LIN {X 0,Y 324.336,Z 494.731,A -85,B 0,C 180,E1 -26772.496,E2 -26772.496} C_VEL
LIN {X 0,Y 334.682,Z 439.584,A -85,B 0,C 180,E1 -26774.316,E2 -26774.316} C_VEL
LIN {X 0,Y 333.314,Z 436.436,A -85,B 0,C 180,E1 -26776.094,E2 -26776.094} C_VEL
LIN {X 0,Y 331.956,Z 433.665,A -85,B 0,C 180,E1 -26778.901,E2 -26778.901} C_VEL
LIN {X 0,Y 331.571,Z 433.329,A -85,B 0,C 180,E1 -26780.673,E2 -26780.673} C_VEL
LIN {X 0,Y 331.565,Z 434.08,A -85,B 0,C 180,E1 -26782.586,E2 -26782.586} C_VEL
LIN {X 0,Y 332.161,Z 436.38,A -85,B 0,C 180,E1 -26784.82,E2 -26784.82} C_VEL
LIN {X 0,Y 333.09,Z 439.465,A -85,B 0,C 180,E1 -26786.646,E2 -26786.646} C_VEL
LIN {X 0,Y 334.002,Z 442.99,A -85,B 0,C 180,E1 -26788.056,E2 -26788.056} C_VEL
LIN {X 0,Y 324.195,Z 494.799,A -85,B 0,C 180,E1 -26789.774,E2 -26789.774} C_VEL
LIN {X 0,Y 320.598,Z 508.539,A -85,B 0,C 180,E1 -26790.375,E2 -26790.375} C_VEL
LIN {X 0,Y 316.075,Z 522.357,A -85,B 0,C 180,E1 -26791.184,E2 -26791.184} C_VEL
LIN {X 0,Y 310.686,Z 536.131,A -85,B 0,C 180,E1 -26792.248,E2 -26792.248} C_VEL
LIN {X 0,Y 304.524,Z 549.185,A -85,B 0,C 180,E1 -26793.534,E2 -26793.534} C_VEL
LIN {X 0,Y 298.181,Z 560.797,A -85,B 0,C 180,E1 -26794.987,E2 -26794.987} C_VEL
LIN {X 0,Y 291.665,Z 571.301,A -85,B 0,C 180,E1 -26796.649,E2 -26796.649} C_VEL
LIN {X 0,Y 285.414,Z 580.164,A -85,B 0,C 180,E1 -26798.4,E2 -26798.4} C_VEL
LIN {X 0,Y 278.653,Z 588.74,A -85,B 0,C 180,E1 -26800.545,E2 -26800.545} C_VEL
LIN {X 0,Y 272.465,Z 595.688,A -85,B 0,C 180,E1 -26802.804,E2 -26802.804} C_VEL
LIN {X 0,Y 266.016,Z 601.972,A -85,B 0,C 180,E1 -26805.514,E2 -26805.514} C_VEL
LIN {X 0,Y 260.17,Z 606.737,A -85,B 0,C 180,E1 -26808.351,E2 -26808.351} C_VEL
LIN {X 0,Y 255.014,Z 610.15,A -85,B 0,C 180,E1 -26811.439,E2 -26811.439} C_VEL
LIN {X 0,Y 252.065,Z 611.627,A -85,B 0,C 180,E1 -26813.618,E2 -26813.618} C_VEL
LIN {X 0,Y 248.579,Z 612.578,A -85,B 0,C 180,E1 -26816.769,E2 -26816.769} C_VEL
LIN {X 0,Y 246.132,Z 612.235,A -85,B 0,C 180,E1 -26820,E2 -26820} C_VEL
LIN {X 0,Y 244.401,Z 610.599,A -85,B 0,C 180,E1 -26823.286,E2 -26823.286} C_VEL
LIN {X 0,Y 243.306,Z 607.613,A -85,B 0,C 180,E1 -26826.612,E2 -26826.612} C_VEL
LIN {X 0,Y 243,Z 603.197,A -85,B 0,C 180,E1 -26829.959,E2 -26829.959} C_VEL
LIN {X 0,Y 242.985,Z 598.806,A -85,B 0,C 180,E1 -26832.486,E2 -26832.486} C_VEL
LIN {X 0,Y 243.239,Z 592.317,A -85,B 0,C 180,E1 -26835.448,E2 -26835.448} C_VEL
LIN {X 0,Y 243.619,Z 584.079,A -85,B 0,C 180,E1 -26838.437,E2 -26838.437} C_VEL
LIN {X 0,Y 244.159,Z 575.362,A -85,B 0,C 180,E1 -26841.014,E2 -26841.014} C_VEL
LIN {X 0,Y 244.883,Z 564.653,A -85,B 0,C 180,E1 -26843.606,E2 -26843.606} C_VEL
LIN {X 0,Y 245.783,Z 553.862,A -85,B 0,C 180,E1 -26845.76,E2 -26845.76} C_VEL
LIN {X 0,Y 246.865,Z 541.033,A -85,B 0,C 180,E1 -26847.87,E2 -26847.87} C_VEL
LIN {X 0,Y 247.927,Z 527.88,A -85,B 0,C 180,E1 -26849.631,E2 -26849.631} C_VEL
LIN {X 0,Y 249.014,Z 513.803,A -85,B 0,C 180,E1 -26851.122,E2 -26851.122} C_VEL
LIN {X 0,Y 250.108,Z 498.529,A -85,B 0,C 180,E1 -26852.359,E2 -26852.359} C_VEL
LIN {X 0,Y 251.001,Z 483.418,A -85,B 0,C 180,E1 -26853.241,E2 -26853.241} C_VEL
LIN {X 0,Y 255.021,Z 389.699,A -85,B 0,C 180,E1 -26857.363,E2 -26857.363} C_VEL
LIN {X 0,Y 252.513,Z 363.65,A -85,B 0,C 180,E1 -26858.616,E2 -26858.616} C_VEL
LIN {X 0,Y 251.535,Z 352.061,A -85,B 0,C 180,E1 -26859.176,E2 -26859.176} C_VEL
LIN {X 0,Y 250.283,Z 346.912,A -85,B 0,C 180,E1 -26859.516,E2 -26859.516} C_VEL
LIN {X 0,Y 246.827,Z 329.605,A -85,B 0,C 180,E1 -26863.64,E2 -26863.64} C_VEL
LIN {X 0,Y 246.163,Z 326.374,A -85,B 0,C 180,E1 -26864.432,E2 -26864.432} C_VEL
LIN {X 0,Y 246.097,Z 326.384,A -85,B 0,C 180,E1 -26869.104,E2 -26869.104} C_VEL
LIN {X 0,Y 246.107,Z 326.385,A -85,B 0,C 180,E1 -26873.292,E2 -26873.292} C_VEL
LIN {X 0,Y 246.115,Z 326.372,A -85,B 0,C 180,E1 -26877.262,E2 -26877.262} C_VEL
LIN {X 0,Y 246.14,Z 326.368,A -85,B 0,C 180,E1 -26881.906,E2 -26881.906} C_VEL
LIN {X 0,Y 246.192,Z 326.378,A -85,B 0,C 180,E1 -26886.523,E2 -26886.523} C_VEL
LIN {X 0,Y 246.258,Z 326.518,A -85,B 0,C 180,E1 -26887.721,E2 -26887.721} C_VEL
LIN {X 0,Y 247.292,Z 329.319,A -85,B 0,C 180,E1 -26887.949,E2 -26887.949} C_VEL
LIN {X 0,Y 255.224,Z 344.588,A -85,B 0,C 180,E1 -26889.436,E2 -26889.436} C_VEL
LIN {X 0,Y 263.934,Z 364.446,A -85,B 0,C 180,E1 -26891.038,E2 -26891.038} C_VEL
LIN {X 0,Y 264.785,Z 366.831,A -85,B 0,C 180,E1 -26891.201,E2 -26891.201} C_VEL
LIN {X 0,Y 261.589,Z 454.014,A -85,B 0,C 180,E1 -26893.517,E2 -26893.517} C_VEL
LIN {X 0,Y 260.624,Z 467.692,A -85,B 0,C 180,E1 -26894.156,E2 -26894.156} C_VEL
LIN {X 0,Y 259.477,Z 480.564,A -85,B 0,C 180,E1 -26895.037,E2 -26895.037} C_VEL
LIN {X 0,Y 257.894,Z 493.809,A -85,B 0,C 180,E1 -26896.248,E2 -26896.248} C_VEL
LIN {X 0,Y 256.075,Z 505.205,A -85,B 0,C 180,E1 -26897.557,E2 -26897.557} C_VEL
LIN {X 0,Y 253.893,Z 517.109,A -85,B 0,C 180,E1 -26899.264,E2 -26899.264} C_VEL
LIN {X 0,Y 251.992,Z 527.921,A -85,B 0,C 180,E1 -26901.202,E2 -26901.202} C_VEL
LIN {X 0,Y 250.122,Z 537.025,A -85,B 0,C 180,E1 -26903.161,E2 -26903.161} C_VEL
LIN {X 0,Y 248.243,Z 546.151,A -85,B 0,C 180,E1 -26905.546,E2 -26905.546} C_VEL
LIN {X 0,Y 246.553,Z 553.781,A -85,B 0,C 180,E1 -26907.961,E2 -26907.961} C_VEL
LIN {X 0,Y 245.444,Z 561.092,A -85,B 0,C 180,E1 -26910.849,E2 -26910.849} C_VEL
LIN {X 0,Y 244.645,Z 566.113,A -85,B 0,C 180,E1 -26913.279,E2 -26913.279} C_VEL
LIN {X 0,Y 243.723,Z 571.419,A -85,B 0,C 180,E1 -26916.597,E2 -26916.597} C_VEL
LIN {X 0,Y 243.365,Z 575.2,A -85,B 0,C 180,E1 -26919.94,E2 -26919.94} C_VEL
LIN {X 0,Y 243.416,Z 576.779,A -85,B 0,C 180,E1 -26921.938,E2 -26921.938} C_VEL
LIN {X 0,Y 243.611,Z 578.262,A -85,B 0,C 180,E1 -26924.993,E2 -26924.993} C_VEL
LIN {X 0,Y 244.447,Z 578.607,A -85,B 0,C 180,E1 -26928.368,E2 -26928.368} C_VEL
LIN {X 0,Y 245.791,Z 577.592,A -85,B 0,C 180,E1 -26931.74,E2 -26931.74} C_VEL
LIN {X 0,Y 247.865,Z 575.178,A -85,B 0,C 180,E1 -26935.075,E2 -26935.075} C_VEL
LIN {X 0,Y 250.574,Z 571.251,A -85,B 0,C 180,E1 -26938.368,E2 -26938.368} C_VEL
LIN {X 0,Y 253.98,Z 565.673,A -85,B 0,C 180,E1 -26941.596,E2 -26941.596} C_VEL
LIN {X 0,Y 257.568,Z 559.306,A -85,B 0,C 180,E1 -26944.348,E2 -26944.348} C_VEL
LIN {X 0,Y 261.631,Z 551.305,A -85,B 0,C 180,E1 -26947.035,E2 -26947.035} C_VEL
LIN {X 0,Y 265.504,Z 542.866,A -85,B 0,C 180,E1 -26949.278,E2 -26949.278} C_VEL
LIN {X 0,Y 269.799,Z 532.633,A -85,B 0,C 180,E1 -26951.448,E2 -26951.448} C_VEL
LIN {X 0,Y 273.597,Z 522.235,A -85,B 0,C 180,E1 -26953.217,E2 -26953.217} C_VEL
LIN {X 0,Y 277.182,Z 510.885,A -85,B 0,C 180,E1 -26954.776,E2 -26954.776} C_VEL
LIN {X 0,Y 280.433,Z 498.58,A -85,B 0,C 180,E1 -26956.123,E2 -26956.123} C_VEL
LIN {X 0,Y 283.166,Z 485.53,A -85,B 0,C 180,E1 -26957.247,E2 -26957.247} C_VEL
LIN {X 0,Y 285.407,Z 471.872,A -85,B 0,C 180,E1 -26958.12,E2 -26958.12} C_VEL
LIN {X 0,Y 286.998,Z 457.659,A -85,B 0,C 180,E1 -26958.759,E2 -26958.759} C_VEL
LIN {X 0,Y 288.327,Z 435.678,A -85,B 0,C 180,E1 -26959.349,E2 -26959.349} C_VEL
LIN {X 0,Y 290.593,Z 394.903,A -85,B 0,C 180,E1 -26960.299,E2 -26960.299} C_VEL
LIN {X 0,Y 285.026,Z 383.377,A -85,B 0,C 180,E1 -26961.787,E2 -26961.787} C_VEL
LIN {X 0,Y 277.938,Z 371.273,A -85,B 0,C 180,E1 -26963.732,E2 -26963.732} C_VEL
LIN {X 0,Y 269.772,Z 358.534,A -85,B 0,C 180,E1 -26966.163,E2 -26966.163} C_VEL
LIN {X 0,Y 263.662,Z 349.923,A -85,B 0,C 180,E1 -26968.131,E2 -26968.131} C_VEL
LIN {X 0,Y 260.517,Z 345.727,A -85,B 0,C 180,E1 -26969.206,E2 -26969.206} C_VEL
LIN {X 0,Y 257.438,Z 341.575,A -85,B 0,C 180,E1 -26970.314,E2 -26970.314} C_VEL
LIN {X 0,Y 254.794,Z 338.233,A -85,B 0,C 180,E1 -26971.303,E2 -26971.303} C_VEL
LIN {X 0,Y 253.958,Z 336.946,A -85,B 0,C 180,E1 -26971.637,E2 -26971.637} C_VEL
LIN {X 0,Y 251.405,Z 334.263,A -85,B 0,C 180,E1 -26972.626,E2 -26972.626} C_VEL
LIN {X 0,Y 250.075,Z 331.865,A -85,B 0,C 180,E1 -26973.211,E2 -26973.211} C_VEL
LIN {X 0,Y 247.587,Z 329.867,A -85,B 0,C 180,E1 -26974.216,E2 -26974.216} C_VEL
LIN {X 0,Y 246.353,Z 327.371,A -85,B 0,C 180,E1 -26974.818,E2 -26974.818} C_VEL
LIN {X 0,Y 246.153,Z 326.379,A -85,B 0,C 180,E1 -26974.985,E2 -26974.985} C_VEL
LIN {X 0,Y 246.241,Z 326.357,A -85,B 0,C 180,E1 -26980.041,E2 -26980.041} C_VEL
LIN {X 0,Y 246.352,Z 326.338,A -85,B 0,C 180,E1 -26985.173,E2 -26985.173} C_VEL
LIN {X 0,Y 246.419,Z 326.329,A -85,B 0,C 180,E1 -26990.18,E2 -26990.18} C_VEL
LIN {X 0,Y 246.664,Z 326.319,A -85,B 0,C 180,E1 -26993.616,E2 -26993.616} C_VEL
LIN {X 0,Y 246.74,Z 326.284,A -85,B 0,C 180,E1 -26996.745,E2 -26996.745} C_VEL
LIN {X 0,Y 246.882,Z 326.281,A -85,B 0,C 180,E1 -27000,E2 -27000} C_VEL
LIN {X 0,Y 246.676,Z 326.314,A -85,B 0,C 180,E1 -27004.887,E2 -27004.887} C_VEL
LIN {X 0,Y 246.504,Z 326.314,A -85,B 0,C 180,E1 -27008.168,E2 -27008.168} C_VEL
LIN {X 0,Y 246.377,Z 326.328,A -85,B 0,C 180,E1 -27013.146,E2 -27013.146} C_VEL
LIN {X 0,Y 246.238,Z 326.35,A -85,B 0,C 180,E1 -27016.527,E2 -27016.527} C_VEL
LIN {X 0,Y 246.239,Z 326.367,A -85,B 0,C 180,E1 -27020.178,E2 -27020.178} C_VEL
LIN {X 0,Y 246.182,Z 326.378,A -85,B 0,C 180,E1 -27024.441,E2 -27024.441} C_VEL
LIN {X 0,Y 246.116,Z 326.383,A -85,B 0,C 180,E1 -27028.935,E2 -27028.935} C_VEL
LIN {X 0,Y 246.158,Z 326.575,A -85,B 0,C 180,E1 -27030.337,E2 -27030.337} C_VEL
LIN {X 0,Y 248.112,Z 332.099,A -85,B 0,C 180,E1 -27034.376,E2 -27034.376} C_VEL
LIN {X 0,Y 249.773,Z 337.188,A -85,B 0,C 180,E1 -27037.671,E2 -27037.671} C_VEL
LIN {X 0,Y 250.499,Z 339.036,A -85,B 0,C 180,E1 -27038.421,E2 -27038.421} C_VEL
LIN {X 0,Y 252.088,Z 343.111,A -85,B 0,C 180,E1 -27039.303,E2 -27039.303} C_VEL
LIN {X 0,Y 255.959,Z 356.555,A -85,B 0,C 180,E1 -27041.169,E2 -27041.169} C_VEL
LIN {X 0,Y 257.972,Z 360.99,A -85,B 0,C 180,E1 -27041.993,E2 -27041.993} C_VEL
LIN {X 0,Y 262.83,Z 369.266,A -85,B 0,C 180,E1 -27043.728,E2 -27043.728} C_VEL
LIN {X 0,Y 269.015,Z 380.503,A -85,B 0,C 180,E1 -27045.79,E2 -27045.79} C_VEL
LIN {X 0,Y 275.663,Z 394.149,A -85,B 0,C 180,E1 -27047.871,E2 -27047.871} C_VEL
LIN {X 0,Y 281.475,Z 407.899,A -85,B 0,C 180,E1 -27049.612,E2 -27049.612} C_VEL
LIN {X 0,Y 283.693,Z 427.748,A -85,B 0,C 180,E1 -27050.754,E2 -27050.754} C_VEL
LIN {X 0,Y 280.723,Z 478.618,A -85,B 0,C 180,E1 -27051.981,E2 -27051.981} C_VEL
LIN {X 0,Y 278.945,Z 493.561,A -85,B 0,C 180,E1 -27052.55,E2 -27052.55} C_VEL
LIN {X 0,Y 276.399,Z 507.618,A -85,B 0,C 180,E1 -27053.342,E2 -27053.342} C_VEL
LIN {X 0,Y 273.137,Z 520.704,A -85,B 0,C 180,E1 -27054.314,E2 -27054.314} C_VEL
LIN {X 0,Y 269.411,Z 533.352,A -85,B 0,C 180,E1 -27055.569,E2 -27055.569} C_VEL
LIN {X 0,Y 265.436,Z 544.887,A -85,B 0,C 180,E1 -27057.031,E2 -27057.031} C_VEL
LIN {X 0,Y 261.709,Z 554.52,A -85,B 0,C 180,E1 -27058.545,E2 -27058.545} C_VEL
LIN {X 0,Y 257.195,Z 565.227,A -85,B 0,C 180,E1 -27060.65,E2 -27060.65} C_VEL
LIN {X 0,Y 252.953,Z 574.104,A -85,B 0,C 180,E1 -27062.818,E2 -27062.818} C_VEL
LIN {X 0,Y 248.616,Z 582.646,A -85,B 0,C 180,E1 -27065.45,E2 -27065.45} C_VEL
LIN {X 0,Y 244.877,Z 589.57,A -85,B 0,C 180,E1 -27068.175,E2 -27068.175} C_VEL
LIN {X 0,Y 241.579,Z 595.839,A -85,B 0,C 180,E1 -27071.406,E2 -27071.406} C_VEL
LIN {X 0,Y 239.033,Z 600.505,A -85,B 0,C 180,E1 -27074.713,E2 -27074.713} C_VEL
LIN {X 0,Y 237.261,Z 603.739,A -85,B 0,C 180,E1 -27078.078,E2 -27078.078} C_VEL
LIN {X 0,Y 236.26,Z 605.64,A -85,B 0,C 180,E1 -27081.48,E2 -27081.48} C_VEL
LIN {X 0,Y 236.139,Z 606.252,A -85,B 0,C 180,E1 -27084.899,E2 -27084.899} C_VEL
LIN {X 0,Y 236.758,Z 605.572,A -85,B 0,C 180,E1 -27088.309,E2 -27088.309} C_VEL
LIN {X 0,Y 236.863,Z 605.464,A -85,B 0,C 180,E1 -27088.839,E2 -27088.839} C_VEL
LIN {X 0,Y 236.642,Z 610.52,A -85,B 0,C 180,E1 -27091.7,E2 -27091.7} C_VEL
LIN {X 0,Y 236.296,Z 614.967,A -85,B 0,C 180,E1 -27095.106,E2 -27095.106} C_VEL
LIN {X 0,Y 236.54,Z 617.99,A -85,B 0,C 180,E1 -27098.519,E2 -27098.519} C_VEL
LIN {X 0,Y 237.781,Z 619.728,A -85,B 0,C 180,E1 -27101.904,E2 -27101.904} C_VEL
LIN {X 0,Y 240.003,Z 620.221,A -85,B 0,C 180,E1 -27105.232,E2 -27105.232} C_VEL
LIN {X 0,Y 243.059,Z 619.47,A -85,B 0,C 180,E1 -27108.485,E2 -27108.485} C_VEL
LIN {X 0,Y 247.046,Z 617.486,A -85,B 0,C 180,E1 -27111.632,E2 -27111.632} C_VEL
LIN {X 0,Y 252.05,Z 614.222,A -85,B 0,C 180,E1 -27114.64,E2 -27114.64} C_VEL
LIN {X 0,Y 257.622,Z 609.641,A -85,B 0,C 180,E1 -27117.534,E2 -27117.534} C_VEL
LIN {X 0,Y 264.117,Z 603.567,A -85,B 0,C 180,E1 -27120.261,E2 -27120.261} C_VEL
LIN {X 0,Y 271.466,Z 595.842,A -85,B 0,C 180,E1 -27122.813,E2 -27122.813} C_VEL
LIN {X 0,Y 278.383,Z 587.587,A -85,B 0,C 180,E1 -27124.923,E2 -27124.923} C_VEL
LIN {X 0,Y 285.87,Z 577.594,A -85,B 0,C 180,E1 -27126.895,E2 -27126.895} C_VEL
LIN {X 0,Y 292.736,Z 567.286,A -85,B 0,C 180,E1 -27128.474,E2 -27128.474} C_VEL
LIN {X 0,Y 299.238,Z 556.134,A -85,B 0,C 180,E1 -27129.854,E2 -27129.854} C_VEL
LIN {X 0,Y 305.485,Z 543.891,A -85,B 0,C 180,E1 -27131.025,E2 -27131.025} C_VEL
LIN {X 0,Y 311.332,Z 530.596,A -85,B 0,C 180,E1 -27132.018,E2 -27132.018} C_VEL
LIN {X 0,Y 316.265,Z 517.205,A -85,B 0,C 180,E1 -27132.776,E2 -27132.776} C_VEL
LIN {X 0,Y 320.797,Z 501.723,A -85,B 0,C 180,E1 -27133.461,E2 -27133.461} C_VEL
LIN {X 0,Y 324.988,Z 481.781,A -85,B 0,C 180,E1 -27134.153,E2 -27134.153} C_VEL
LIN {X 0,Y 332.174,Z 444.696,A -85,B 0,C 180,E1 -27135.374,E2 -27135.374} C_VEL
LIN {X 0,Y 331.261,Z 442.694,A -85,B 0,C 180,E1 -27136.763,E2 -27136.763} C_VEL
LIN {X 0,Y 330.257,Z 440.394,A -85,B 0,C 180,E1 -27139.321,E2 -27139.321} C_VEL
LIN {X 0,Y 329.944,Z 440.521,A -85,B 0,C 180,E1 -27141.769,E2 -27141.769} C_VEL
LIN {X 0,Y 330.263,Z 442.496,A -85,B 0,C 180,E1 -27144.061,E2 -27144.061} C_VEL
LIN {X 0,Y 330.815,Z 444.6,A -85,B 0,C 180,E1 -27145.522,E2 -27145.522} C_VEL
LIN {X 0,Y 331.491,Z 447.394,A -85,B 0,C 180,E1 -27146.868,E2 -27146.868} C_VEL
LIN {X 0,Y 331.544,Z 447.912,A -85,B 0,C 180,E1 -27147.019,E2 -27147.019} C_VEL
LIN {X 0,Y 322.252,Z 495.042,A -85,B 0,C 180,E1 -27148.556,E2 -27148.556} C_VEL
LIN {X 0,Y 318.393,Z 509.201,A -85,B 0,C 180,E1 -27149.169,E2 -27149.169} C_VEL
LIN {X 0,Y 313.488,Z 523.557,A -85,B 0,C 180,E1 -27150.004,E2 -27150.004} C_VEL
LIN {X 0,Y 307.748,Z 537.416,A -85,B 0,C 180,E1 -27151.075,E2 -27151.075} C_VEL
LIN {X 0,Y 300.838,Z 551.253,A -85,B 0,C 180,E1 -27152.456,E2 -27152.456} C_VEL
LIN {X 0,Y 294.321,Z 562.449,A -85,B 0,C 180,E1 -27153.879,E2 -27153.879} C_VEL
LIN {X 0,Y 287.545,Z 572.735,A -85,B 0,C 180,E1 -27155.537,E2 -27155.537} C_VEL
LIN {X 0,Y 280.861,Z 581.621,A -85,B 0,C 180,E1 -27157.338,E2 -27157.338} C_VEL
LIN {X 0,Y 274.007,Z 589.691,A -85,B 0,C 180,E1 -27159.421,E2 -27159.421} C_VEL
LIN {X 0,Y 267.52,Z 596.488,A -85,B 0,C 180,E1 -27161.688,E2 -27161.688} C_VEL
LIN {X 0,Y 260.74,Z 602.634,A -85,B 0,C 180,E1 -27164.417,E2 -27164.417} C_VEL
LIN {X 0,Y 254.608,Z 607.263,A -85,B 0,C 180,E1 -27167.286,E2 -27167.286} C_VEL
LIN {X 0,Y 249.313,Z 610.449,A -85,B 0,C 180,E1 -27170.295,E2 -27170.295} C_VEL
LIN {X 0,Y 244.945,Z 612.283,A -85,B 0,C 180,E1 -27173.432,E2 -27173.432} C_VEL
LIN {X 0,Y 241.432,Z 612.82,A -85,B 0,C 180,E1 -27176.674,E2 -27176.674} C_VEL
LIN {X 0,Y 238.962,Z 612.075,A -85,B 0,C 180,E1 -27180,E2 -27180} C_VEL
LIN {X 0,Y 237.236,Z 610.044,A -85,B 0,C 180,E1 -27183.385,E2 -27183.385} C_VEL
LIN {X 0,Y 236.193,Z 606.65,A -85,B 0,C 180,E1 -27186.813,E2 -27186.813} C_VEL
LIN {X 0,Y 235.943,Z 601.793,A -85,B 0,C 180,E1 -27190.26,E2 -27190.26} C_VEL
LIN {X 0,Y 235.966,Z 597.046,A -85,B 0,C 180,E1 -27192.864,E2 -27192.864} C_VEL
LIN {X 0,Y 236.283,Z 590.09,A -85,B 0,C 180,E1 -27195.915,E2 -27195.915} C_VEL
LIN {X 0,Y 236.657,Z 582.174,A -85,B 0,C 180,E1 -27198.707,E2 -27198.707} C_VEL
LIN {X 0,Y 237.175,Z 573.576,A -85,B 0,C 180,E1 -27201.209,E2 -27201.209} C_VEL
LIN {X 0,Y 237.977,Z 562.146,A -85,B 0,C 180,E1 -27203.949,E2 -27203.949} C_VEL
LIN {X 0,Y 238.967,Z 550.077,A -85,B 0,C 180,E1 -27206.317,E2 -27206.317} C_VEL
LIN {X 0,Y 240.059,Z 537.136,A -85,B 0,C 180,E1 -27208.366,E2 -27208.366} C_VEL
LIN {X 0,Y 241.147,Z 523.888,A -85,B 0,C 180,E1 -27210.069,E2 -27210.069} C_VEL
LIN {X 0,Y 242.168,Z 509.966,A -85,B 0,C 180,E1 -27211.496,E2 -27211.496} C_VEL
LIN {X 0,Y 243.2,Z 495.468,A -85,B 0,C 180,E1 -27212.624,E2 -27212.624} C_VEL
LIN {X 0,Y 244.086,Z 479.061,A -85,B 0,C 180,E1 -27213.53,E2 -27213.53} C_VEL
LIN {X 0,Y 247.981,Z 390.378,A -85,B 0,C 180,E1 -27217.561,E2 -27217.561} C_VEL
LIN {X 0,Y 245.383,Z 362.456,A -85,B 0,C 180,E1 -27218.948,E2 -27218.948} C_VEL
LIN {X 0,Y 244.574,Z 353.328,A -85,B 0,C 180,E1 -27219.407,E2 -27219.407} C_VEL
LIN {X 0,Y 243.104,Z 347.07,A -85,B 0,C 180,E1 -27219.816,E2 -27219.816} C_VEL
LIN {X 0,Y 239.64,Z 329.856,A -85,B 0,C 180,E1 -27224.001,E2 -27224.001} C_VEL
LIN {X 0,Y 239.115,Z 327.25,A -85,B 0,C 180,E1 -27224.671,E2 -27224.671} C_VEL
LIN {X 0,Y 239.062,Z 327.259,A -85,B 0,C 180,E1 -27229.86,E2 -27229.86} C_VEL
LIN {X 0,Y 239.033,Z 327.258,A -85,B 0,C 180,E1 -27234.117,E2 -27234.117} C_VEL
LIN {X 0,Y 239.084,Z 327.256,A -85,B 0,C 180,E1 -27238.17,E2 -27238.17} C_VEL
LIN {X 0,Y 239.101,Z 327.244,A -85,B 0,C 180,E1 -27242.045,E2 -27242.045} C_VEL
LIN {X 0,Y 239.161,Z 327.274,A -85,B 0,C 180,E1 -27246.775,E2 -27246.775} C_VEL
LIN {X 0,Y 240.225,Z 330.204,A -85,B 0,C 180,E1 -27247.025,E2 -27247.025} C_VEL
LIN {X 0,Y 247.828,Z 344.438,A -85,B 0,C 180,E1 -27248.515,E2 -27248.515} C_VEL
LIN {X 0,Y 256.291,Z 363.144,A -85,B 0,C 180,E1 -27250.143,E2 -27250.143} C_VEL
LIN {X 0,Y 258.304,Z 368.174,A -85,B 0,C 180,E1 -27250.529,E2 -27250.529} C_VEL
LIN {X 0,Y 255.131,Z 454.419,A -85,B 0,C 180,E1 -27252.882,E2 -27252.882} C_VEL
LIN {X 0,Y 254.127,Z 468.101,A -85,B 0,C 180,E1 -27253.534,E2 -27253.534} C_VEL
LIN {X 0,Y 252.798,Z 482.095,A -85,B 0,C 180,E1 -27254.529,E2 -27254.529} C_VEL
LIN {X 0,Y 251.077,Z 495.959,A -85,B 0,C 180,E1 -27255.867,E2 -27255.867} C_VEL
LIN {X 0,Y 248.941,Z 508.449,A -85,B 0,C 180,E1 -27257.401,E2 -27257.401} C_VEL
LIN {X 0,Y 246.757,Z 519.848,A -85,B 0,C 180,E1 -27259.157,E2 -27259.157} C_VEL
LIN {X 0,Y 245.004,Z 529.301,A -85,B 0,C 180,E1 -27260.949,E2 -27260.949} C_VEL
LIN {X 0,Y 242.7,Z 539.876,A -85,B 0,C 180,E1 -27263.367,E2 -27263.367} C_VEL
LIN {X 0,Y 240.884,Z 548.588,A -85,B 0,C 180,E1 -27265.827,E2 -27265.827} C_VEL
LIN {X 0,Y 239.242,Z 555.863,A -85,B 0,C 180,E1 -27268.318,E2 -27268.318} C_VEL
LIN {X 0,Y 238.204,Z 562.68,A -85,B 0,C 180,E1 -27271.211,E2 -27271.211} C_VEL
LIN {X 0,Y 237.237,Z 568.335,A -85,B 0,C 180,E1 -27274.229,E2 -27274.229} C_VEL
LIN {X 0,Y 236.448,Z 573.187,A -85,B 0,C 180,E1 -27277.656,E2 -27277.656} C_VEL
LIN {X 0,Y 236.267,Z 575.802,A -85,B 0,C 180,E1 -27280.242,E2 -27280.242} C_VEL
LIN {X 0,Y 236.385,Z 578.103,A -85,B 0,C 180,E1 -27283.708,E2 -27283.708} C_VEL
LIN {X 0,Y 236.982,Z 579.048,A -85,B 0,C 180,E1 -27287.187,E2 -27287.187} C_VEL
LIN {X 0,Y 238.207,Z 578.633,A -85,B 0,C 180,E1 -27290.657,E2 -27290.657} C_VEL
LIN {X 0,Y 240.027,Z 576.841,A -85,B 0,C 180,E1 -27294.109,E2 -27294.109} C_VEL
LIN {X 0,Y 242.596,Z 573.572,A -85,B 0,C 180,E1 -27297.509,E2 -27297.509} C_VEL
LIN {X 0,Y 245.841,Z 568.734,A -85,B 0,C 180,E1 -27300.849,E2 -27300.849} C_VEL
LIN {X 0,Y 248.786,Z 564.008,A -85,B 0,C 180,E1 -27303.294,E2 -27303.294} C_VEL
LIN {X 0,Y 252.989,Z 556.513,A -85,B 0,C 180,E1 -27306.278,E2 -27306.278} C_VEL
LIN {X 0,Y 257.101,Z 548.39,A -85,B 0,C 180,E1 -27308.795,E2 -27308.795} C_VEL
LIN {X 0,Y 261.2,Z 539.516,A -85,B 0,C 180,E1 -27310.984,E2 -27310.984} C_VEL
LIN {X 0,Y 265.133,Z 530.093,A -85,B 0,C 180,E1 -27312.859,E2 -27312.859} C_VEL
LIN {X 0,Y 269.128,Z 519.084,A -85,B 0,C 180,E1 -27314.639,E2 -27314.639} C_VEL
LIN {X 0,Y 272.872,Z 506.946,A -85,B 0,C 180,E1 -27316.209,E2 -27316.209} C_VEL
LIN {X 0,Y 275.866,Z 495.22,A -85,B 0,C 180,E1 -27317.414,E2 -27317.414} C_VEL
LIN {X 0,Y 278.671,Z 481.327,A -85,B 0,C 180,E1 -27318.527,E2 -27318.527} C_VEL
LIN {X 0,Y 280.812,Z 467.022,A -85,B 0,C 180,E1 -27319.347,E2 -27319.347} C_VEL
LIN {X 0,Y 282.152,Z 453.648,A -85,B 0,C 180,E1 -27319.864,E2 -27319.864} C_VEL
LIN {X 0,Y 285.374,Z 397.385,A -85,B 0,C 180,E1 -27321.224,E2 -27321.224} C_VEL
LIN {X 0,Y 280.292,Z 386.884,A -85,B 0,C 180,E1 -27322.643,E2 -27322.643} C_VEL
LIN {X 0,Y 272.88,Z 374.249,A -85,B 0,C 180,E1 -27324.778,E2 -27324.778} C_VEL
LIN {X 0,Y 265.612,Z 362.906,A -85,B 0,C 180,E1 -27327.05,E2 -27327.05} C_VEL
LIN {X 0,Y 260.015,Z 355.002,A -85,B 0,C 180,E1 -27328.933,E2 -27328.933} C_VEL
LIN {X 0,Y 256.903,Z 350.768,A -85,B 0,C 180,E1 -27330.047,E2 -27330.047} C_VEL
LIN {X 0,Y 254.324,Z 347.231,A -85,B 0,C 180,E1 -27331.019,E2 -27331.019} C_VEL
LIN {X 0,Y 251.511,Z 343.38,A -85,B 0,C 180,E1 -27332.129,E2 -27332.129} C_VEL
LIN {X 0,Y 248.474,Z 339.882,A -85,B 0,C 180,E1 -27333.359,E2 -27333.359} C_VEL
LIN {X 0,Y 247.369,Z 338.074,A -85,B 0,C 180,E1 -27333.854,E2 -27333.854} C_VEL
LIN {X 0,Y 244.809,Z 335.604,A -85,B 0,C 180,E1 -27334.952,E2 -27334.952} C_VEL
LIN {X 0,Y 243.284,Z 332.858,A -85,B 0,C 180,E1 -27335.709,E2 -27335.709} C_VEL
LIN {X 0,Y 240.736,Z 330.955,A -85,B 0,C 180,E1 -27336.872,E2 -27336.872} C_VEL
LIN {X 0,Y 239.49,Z 328.827,A -85,B 0,C 180,E1 -27337.54,E2 -27337.54} C_VEL
LIN {X 0,Y 239.114,Z 327.246,A -85,B 0,C 180,E1 -27337.843,E2 -27337.843} C_VEL
LIN {X 0,Y 239.156,Z 327.233,A -85,B 0,C 180,E1 -27341.206,E2 -27341.206} C_VEL
LIN {X 0,Y 239.284,Z 327.219,A -85,B 0,C 180,E1 -27344.995,E2 -27344.995} C_VEL
LIN {X 0,Y 239.367,Z 327.209,A -85,B 0,C 180,E1 -27349.888,E2 -27349.888} C_VEL
LIN {X 0,Y 239.641,Z 327.193,A -85,B 0,C 180,E1 -27353.563,E2 -27353.563} C_VEL
LIN {X 0,Y 239.709,Z 327.159,A -85,B 0,C 180,E1 -27356.65,E2 -27356.65} C_VEL
LIN {X 0,Y 239.847,Z 327.157,A -85,B 0,C 180,E1 -27360,E2 -27360} C_VEL
LIN {X 0,Y 239.711,Z 327.167,A -85,B 0,C 180,E1 -27363.35,E2 -27363.35} C_VEL
LIN {X 0,Y 239.603,Z 327.172,A -85,B 0,C 180,E1 -27366.715,E2 -27366.715} C_VEL
LIN {X 0,Y 239.349,Z 327.204,A -85,B 0,C 180,E1 -27371.821,E2 -27371.821} C_VEL
LIN {X 0,Y 239.28,Z 327.233,A -85,B 0,C 180,E1 -27375.275,E2 -27375.275} C_VEL
LIN {X 0,Y 239.175,Z 327.241,A -85,B 0,C 180,E1 -27380.575,E2 -27380.575} C_VEL
LIN {X 0,Y 239.12,Z 327.254,A -85,B 0,C 180,E1 -27384.772,E2 -27384.772} C_VEL
LIN {X 0,Y 239.131,Z 327.352,A -85,B 0,C 180,E1 -27387.71,E2 -27387.71} C_VEL
LIN {X 0,Y 241.226,Z 333.465,A -85,B 0,C 180,E1 -27392.65,E2 -27392.65} C_VEL
LIN {X 0,Y 242.742,Z 337.837,A -85,B 0,C 180,E1 -27395.611,E2 -27395.611} C_VEL
LIN {X 0,Y 246.06,Z 342.861,A -85,B 0,C 180,E1 -27397.173,E2 -27397.173} C_VEL
LIN {X 0,Y 247.675,Z 344.955,A -85,B 0,C 180,E1 -27397.873,E2 -27397.873} C_VEL
LIN {X 0,Y 251.111,Z 350.075,A -85,B 0,C 180,E1 -27399.325,E2 -27399.325} C_VEL
LIN {X 0,Y 256.089,Z 357.941,A -85,B 0,C 180,E1 -27401.289,E2 -27401.289} C_VEL
LIN {X 0,Y 257.972,Z 360.99,A -85,B 0,C 180,E1 -27401.993,E2 -27401.993} C_VEL
LIN {X 0,Y 260.017,Z 365.229,A -85,B 0,C 180,E1 -27402.774,E2 -27402.774} C_VEL
LIN {X 0,Y 261.538,Z 370.158,A -85,B 0,C 180,E1 -27403.415,E2 -27403.415} C_VEL
LIN {X 0,Y 265.001,Z 384.136,A -85,B 0,C 180,E1 -27404.93,E2 -27404.93} C_VEL
LIN {X 0,Y 266.209,Z 387.353,A -85,B 0,C 180,E1 -27405.37,E2 -27405.37} C_VEL
LIN {X 0,Y 272.772,Z 401.414,A -85,B 0,C 180,E1 -27407.499,E2 -27407.499} C_VEL
LIN {X 0,Y 276.741,Z 411.518,A -85,B 0,C 180,E1 -27408.754,E2 -27408.754} C_VEL
LIN {X 0,Y 278.598,Z 429.253,A -85,B 0,C 180,E1 -27409.789,E2 -27409.789} C_VEL
LIN {X 0,Y 275.483,Z 479.381,A -85,B 0,C 180,E1 -27411.007,E2 -27411.007} C_VEL
LIN {X 0,Y 273.639,Z 493.819,A -85,B 0,C 180,E1 -27411.577,E2 -27411.577} C_VEL
LIN {X 0,Y 271.024,Z 507.702,A -85,B 0,C 180,E1 -27412.374,E2 -27412.374} C_VEL
LIN {X 0,Y 267.417,Z 521.559,A -85,B 0,C 180,E1 -27413.429,E2 -27413.429} C_VEL
LIN {X 0,Y 263.625,Z 533.958,A -85,B 0,C 180,E1 -27414.703,E2 -27414.703} C_VEL
LIN {X 0,Y 259.082,Z 546.483,A -85,B 0,C 180,E1 -27416.347,E2 -27416.347} C_VEL
LIN {X 0,Y 254.92,Z 556.747,A -85,B 0,C 180,E1 -27418.072,E2 -27418.072} C_VEL
LIN {X 0,Y 250.291,Z 567.002,A -85,B 0,C 180,E1 -27420.22,E2 -27420.22} C_VEL
LIN {X 0,Y 245.971,Z 575.519,A -85,B 0,C 180,E1 -27422.44,E2 -27422.44} C_VEL
LIN {X 0,Y 241.572,Z 583.701,A -85,B 0,C 180,E1 -27425.143,E2 -27425.143} C_VEL
LIN {X 0,Y 238.275,Z 589.47,A -85,B 0,C 180,E1 -27427.538,E2 -27427.538} C_VEL
LIN {X 0,Y 234.836,Z 595.651,A -85,B 0,C 180,E1 -27430.851,E2 -27430.851} C_VEL
LIN {X 0,Y 232.15,Z 600.243,A -85,B 0,C 180,E1 -27434.248,E2 -27434.248} C_VEL
LIN {X 0,Y 230.282,Z 603.42,A -85,B 0,C 180,E1 -27437.711,E2 -27437.711} C_VEL
LIN {X 0,Y 229.214,Z 605.265,A -85,B 0,C 180,E1 -27441.216,E2 -27441.216} C_VEL
LIN {X 0,Y 229.041,Z 605.821,A -85,B 0,C 180,E1 -27444.74,E2 -27444.74} C_VEL
LIN {X 0,Y 229.655,Z 605.086,A -85,B 0,C 180,E1 -27448.257,E2 -27448.257} C_VEL
LIN {X 0,Y 229.871,Z 604.838,A -85,B 0,C 180,E1 -27449.24,E2 -27449.24} C_VEL
LIN {X 0,Y 229.653,Z 609.278,A -85,B 0,C 180,E1 -27451.752,E2 -27451.752} C_VEL
LIN {X 0,Y 229.314,Z 613.971,A -85,B 0,C 180,E1 -27455.262,E2 -27455.262} C_VEL
LIN {X 0,Y 229.544,Z 617.232,A -85,B 0,C 180,E1 -27458.78,E2 -27458.78} C_VEL
LIN {X 0,Y 230.839,Z 619.23,A -85,B 0,C 180,E1 -27462.267,E2 -27462.267} C_VEL
LIN {X 0,Y 233.153,Z 619.992,A -85,B 0,C 180,E1 -27465.691,E2 -27465.691} C_VEL
LIN {X 0,Y 236.334,Z 619.526,A -85,B 0,C 180,E1 -27469.031,E2 -27469.031} C_VEL
LIN {X 0,Y 240.476,Z 617.84,A -85,B 0,C 180,E1 -27472.255,E2 -27472.255} C_VEL
LIN {X 0,Y 245.643,Z 614.89,A -85,B 0,C 180,E1 -27475.327,E2 -27475.327} C_VEL
LIN {X 0,Y 251.422,Z 610.655,A -85,B 0,C 180,E1 -27478.273,E2 -27478.273} C_VEL
LIN {X 0,Y 258.128,Z 605.007,A -85,B 0,C 180,E1 -27481.04,E2 -27481.04} C_VEL
LIN {X 0,Y 265.683,Z 597.785,A -85,B 0,C 180,E1 -27483.621,E2 -27483.621} C_VEL
LIN {X 0,Y 273.863,Z 588.755,A -85,B 0,C 180,E1 -27486.037,E2 -27486.037} C_VEL
LIN {X 0,Y 281.603,Z 579.054,A -85,B 0,C 180,E1 -27488.001,E2 -27488.001} C_VEL
LIN {X 0,Y 288.679,Z 569.115,A -85,B 0,C 180,E1 -27489.567,E2 -27489.567} C_VEL
LIN {X 0,Y 296.006,Z 557.336,A -85,B 0,C 180,E1 -27491.049,E2 -27491.049} C_VEL
LIN {X 0,Y 303.024,Z 544.289,A -85,B 0,C 180,E1 -27492.295,E2 -27492.295} C_VEL
LIN {X 0,Y 309.136,Z 530.975,A -85,B 0,C 180,E1 -27493.271,E2 -27493.271} C_VEL
LIN {X 0,Y 314.7,Z 516.399,A -85,B 0,C 180,E1 -27494.074,E2 -27494.074} C_VEL
LIN {X 0,Y 319.497,Z 500.196,A -85,B 0,C 180,E1 -27494.769,E2 -27494.769} C_VEL
LIN {X 0,Y 324.264,Z 477.875,A -85,B 0,C 180,E1 -27495.505,E2 -27495.505} C_VEL
LIN {X 0,Y 329.836,Z 450.121,A -85,B 0,C 180,E1 -27496.418,E2 -27496.418} C_VEL
LIN {X 0,Y 328.712,Z 447.44,A -85,B 0,C 180,E1 -27499.089,E2 -27499.089} C_VEL
LIN {X 0,Y 328.339,Z 447.28,A -85,B 0,C 180,E1 -27501.355,E2 -27501.355} C_VEL
LIN {X 0,Y 328.513,Z 448.861,A -85,B 0,C 180,E1 -27503.512,E2 -27503.512} C_VEL
LIN {X 0,Y 329.029,Z 451.267,A -85,B 0,C 180,E1 -27505.247,E2 -27505.247} C_VEL
LIN {X 0,Y 329.341,Z 452.534,A -85,B 0,C 180,E1 -27505.933,E2 -27505.933} C_VEL
LIN {X 0,Y 320.454,Z 495.837,A -85,B 0,C 180,E1 -27507.342,E2 -27507.342} C_VEL
LIN {X 0,Y 316.574,Z 509.532,A -85,B 0,C 180,E1 -27507.926,E2 -27507.926} C_VEL
LIN {X 0,Y 311.671,Z 523.409,A -85,B 0,C 180,E1 -27508.707,E2 -27508.707} C_VEL
LIN {X 0,Y 305.781,Z 537.184,A -85,B 0,C 180,E1 -27509.738,E2 -27509.738} C_VEL
LIN {X 0,Y 298.682,Z 550.935,A -85,B 0,C 180,E1 -27511.074,E2 -27511.074} C_VEL
LIN {X 0,Y 291.69,Z 562.494,A -85,B 0,C 180,E1 -27512.503,E2 -27512.503} C_VEL
LIN {X 0,Y 284.761,Z 572.61,A -85,B 0,C 180,E1 -27514.112,E2 -27514.112} C_VEL
LIN {X 0,Y 277.928,Z 581.311,A -85,B 0,C 180,E1 -27515.824,E2 -27515.824} C_VEL
LIN {X 0,Y 270.517,Z 589.662,A -85,B 0,C 180,E1 -27517.948,E2 -27517.948} C_VEL
LIN {X 0,Y 264.602,Z 595.615,A -85,B 0,C 180,E1 -27519.871,E2 -27519.871} C_VEL
LIN {X 0,Y 257.281,Z 602,A -85,B 0,C 180,E1 -27522.574,E2 -27522.574} C_VEL
LIN {X 0,Y 250.709,Z 606.813,A -85,B 0,C 180,E1 -27525.437,E2 -27525.437} C_VEL
LIN {X 0,Y 244.855,Z 610.209,A -85,B 0,C 180,E1 -27528.449,E2 -27528.449} C_VEL
LIN {X 0,Y 239.937,Z 612.251,A -85,B 0,C 180,E1 -27531.607,E2 -27531.607} C_VEL
LIN {X 0,Y 235.925,Z 612.999,A -85,B 0,C 180,E1 -27534.89,E2 -27534.89} C_VEL
LIN {X 0,Y 232.908,Z 612.472,A -85,B 0,C 180,E1 -27538.277,E2 -27538.277} C_VEL
LIN {X 0,Y 230.855,Z 610.682,A -85,B 0,C 180,E1 -27541.739,E2 -27541.739} C_VEL
LIN {X 0,Y 229.518,Z 607.574,A -85,B 0,C 180,E1 -27545.253,E2 -27545.253} C_VEL
LIN {X 0,Y 228.95,Z 603.063,A -85,B 0,C 180,E1 -27548.799,E2 -27548.799} C_VEL
LIN {X 0,Y 228.914,Z 598.174,A -85,B 0,C 180,E1 -27551.702,E2 -27551.702} C_VEL
LIN {X 0,Y 229.139,Z 591.032,A -85,B 0,C 180,E1 -27555.06,E2 -27555.06} C_VEL
LIN {X 0,Y 229.481,Z 583.816,A -85,B 0,C 180,E1 -27557.772,E2 -27557.772} C_VEL
LIN {X 0,Y 229.99,Z 575.054,A -85,B 0,C 180,E1 -27560.502,E2 -27560.502} C_VEL
LIN {X 0,Y 230.554,Z 566.247,A -85,B 0,C 180,E1 -27562.79,E2 -27562.79} C_VEL
LIN {X 0,Y 231.474,Z 554.62,A -85,B 0,C 180,E1 -27565.304,E2 -27565.304} C_VEL
LIN {X 0,Y 232.587,Z 541.7,A -85,B 0,C 180,E1 -27567.582,E2 -27567.582} C_VEL
LIN {X 0,Y 233.674,Z 528.697,A -85,B 0,C 180,E1 -27569.45,E2 -27569.45} C_VEL
LIN {X 0,Y 234.733,Z 515.442,A -85,B 0,C 180,E1 -27570.98,E2 -27570.98} C_VEL
LIN {X 0,Y 235.802,Z 500.327,A -85,B 0,C 180,E1 -27572.323,E2 -27572.323} C_VEL
LIN {X 0,Y 236.756,Z 485.061,A -85,B 0,C 180,E1 -27573.31,E2 -27573.31} C_VEL
LIN {X 0,Y 240.958,Z 391.001,A -85,B 0,C 180,E1 -27577.763,E2 -27577.763} C_VEL
LIN {X 0,Y 238.4,Z 363.366,A -85,B 0,C 180,E1 -27579.179,E2 -27579.179} C_VEL
LIN {X 0,Y 237.651,Z 354.55,A -85,B 0,C 180,E1 -27579.635,E2 -27579.635} C_VEL
LIN {X 0,Y 235.917,Z 347.305,A -85,B 0,C 180,E1 -27580.089,E2 -27580.089} C_VEL
LIN {X 0,Y 232.509,Z 330.339,A -85,B 0,C 180,E1 -27584.313,E2 -27584.313} C_VEL
LIN {X 0,Y 232.077,Z 328.125,A -85,B 0,C 180,E1 -27584.896,E2 -27584.896} C_VEL
LIN {X 0,Y 231.995,Z 328.141,A -85,B 0,C 180,E1 -27589.008,E2 -27589.008} C_VEL
LIN {X 0,Y 231.999,Z 328.143,A -85,B 0,C 180,E1 -27592.851,E2 -27592.851} C_VEL
LIN {X 0,Y 231.987,Z 328.128,A -85,B 0,C 180,E1 -27597.075,E2 -27597.075} C_VEL
LIN {X 0,Y 232.036,Z 328.127,A -85,B 0,C 180,E1 -27601.115,E2 -27601.115} C_VEL
LIN {X 0,Y 232.123,Z 328.127,A -85,B 0,C 180,E1 -27605.748,E2 -27605.748} C_VEL
LIN {X 0,Y 233.082,Z 330.937,A -85,B 0,C 180,E1 -27606.019,E2 -27606.019} C_VEL
LIN {X 0,Y 237.727,Z 339.222,A -85,B 0,C 180,E1 -27606.985,E2 -27606.985} C_VEL
LIN {X 0,Y 244.83,Z 353.404,A -85,B 0,C 180,E1 -27608.425,E2 -27608.425} C_VEL
LIN {X 0,Y 252.034,Z 370.243,A -85,B 0,C 180,E1 -27609.867,E2 -27609.867} C_VEL
LIN {X 0,Y 248.693,Z 454.834,A -85,B 0,C 180,E1 -27612.213,E2 -27612.213} C_VEL
LIN {X 0,Y 247.663,Z 468.51,A -85,B 0,C 180,E1 -27612.88,E2 -27612.88} C_VEL
LIN {X 0,Y 246.281,Z 482.504,A -85,B 0,C 180,E1 -27613.897,E2 -27613.897} C_VEL
LIN {X 0,Y 244.508,Z 496.365,A -85,B 0,C 180,E1 -27615.267,E2 -27615.267} C_VEL
LIN {X 0,Y 242.298,Z 508.857,A -85,B 0,C 180,E1 -27616.837,E2 -27616.837} C_VEL
LIN {X 0,Y 240.042,Z 520.257,A -85,B 0,C 180,E1 -27618.636,E2 -27618.636} C_VEL
LIN {X 0,Y 238.027,Z 530.68,A -85,B 0,C 180,E1 -27620.682,E2 -27620.682} C_VEL
LIN {X 0,Y 235.64,Z 541.102,A -85,B 0,C 180,E1 -27623.167,E2 -27623.167} C_VEL
LIN {X 0,Y 233.811,Z 549.675,A -85,B 0,C 180,E1 -27625.701,E2 -27625.701} C_VEL
LIN {X 0,Y 232.157,Z 556.83,A -85,B 0,C 180,E1 -27628.267,E2 -27628.267} C_VEL
LIN {X 0,Y 231.181,Z 562.997,A -85,B 0,C 180,E1 -27630.985,E2 -27630.985} C_VEL
LIN {X 0,Y 230.092,Z 569.109,A -85,B 0,C 180,E1 -27634.36,E2 -27634.36} C_VEL
LIN {X 0,Y 229.443,Z 572.791,A -85,B 0,C 180,E1 -27637.01,E2 -27637.01} C_VEL
LIN {X 0,Y 229.18,Z 576.404,A -85,B 0,C 180,E1 -27640.562,E2 -27640.562} C_VEL
LIN {X 0,Y 229.338,Z 578.627,A -85,B 0,C 180,E1 -27644.138,E2 -27644.138} C_VEL
LIN {X 0,Y 230.047,Z 579.491,A -85,B 0,C 180,E1 -27647.722,E2 -27647.722} C_VEL
LIN {X 0,Y 231.384,Z 578.993,A -85,B 0,C 180,E1 -27651.296,E2 -27651.296} C_VEL
LIN {X 0,Y 233.371,Z 577.089,A -85,B 0,C 180,E1 -27654.842,E2 -27654.842} C_VEL
LIN {X 0,Y 236.112,Z 573.723,A -85,B 0,C 180,E1 -27658.331,E2 -27658.331} C_VEL
LIN {X 0,Y 239.549,Z 568.795,A -85,B 0,C 180,E1 -27661.752,E2 -27661.752} C_VEL
LIN {X 0,Y 242.687,Z 563.973,A -85,B 0,C 180,E1 -27664.245,E2 -27664.245} C_VEL
LIN {X 0,Y 246.9,Z 556.735,A -85,B 0,C 180,E1 -27667.158,E2 -27667.158} C_VEL
LIN {X 0,Y 251.416,Z 548.132,A -85,B 0,C 180,E1 -27669.844,E2 -27669.844} C_VEL
LIN {X 0,Y 256.24,Z 537.957,A -85,B 0,C 180,E1 -27672.322,E2 -27672.322} C_VEL
LIN {X 0,Y 260.592,Z 527.477,A -85,B 0,C 180,E1 -27674.329,E2 -27674.329} C_VEL
LIN {X 0,Y 264.673,Z 516.215,A -85,B 0,C 180,E1 -27676.05,E2 -27676.05} C_VEL
LIN {X 0,Y 268.298,Z 504.278,A -85,B 0,C 180,E1 -27677.514,E2 -27677.514} C_VEL
LIN {X 0,Y 271.621,Z 490.743,A -85,B 0,C 180,E1 -27678.816,E2 -27678.816} C_VEL
LIN {X 0,Y 274.1,Z 477.807,A -85,B 0,C 180,E1 -27679.761,E2 -27679.761} C_VEL
LIN {X 0,Y 276.061,Z 463.671,A -85,B 0,C 180,E1 -27680.513,E2 -27680.513} C_VEL
LIN {X 0,Y 277.357,Z 449.239,A -85,B 0,C 180,E1 -27680.995,E2 -27680.995} C_VEL
LIN {X 0,Y 280.157,Z 399.699,A -85,B 0,C 180,E1 -27682.205,E2 -27682.205} C_VEL
LIN {X 0,Y 275.787,Z 390.813,A -85,B 0,C 180,E1 -27683.476,E2 -27683.476} C_VEL
LIN {X 0,Y 268.719,Z 378.572,A -85,B 0,C 180,E1 -27685.612,E2 -27685.612} C_VEL
LIN {X 0,Y 261.602,Z 367.334,A -85,B 0,C 180,E1 -27687.941,E2 -27687.941} C_VEL
LIN {X 0,Y 254.574,Z 357.312,A -85,B 0,C 180,E1 -27690.457,E2 -27690.457} C_VEL
LIN {X 0,Y 250.87,Z 352.416,A -85,B 0,C 180,E1 -27691.891,E2 -27691.891} C_VEL
LIN {X 0,Y 248.024,Z 348.621,A -85,B 0,C 180,E1 -27693.062,E2 -27693.062} C_VEL
LIN {X 0,Y 245.229,Z 344.884,A -85,B 0,C 180,E1 -27694.277,E2 -27694.277} C_VEL
LIN {X 0,Y 241.832,Z 340.941,A -85,B 0,C 180,E1 -27695.825,E2 -27695.825} C_VEL
LIN {X 0,Y 240.667,Z 339.123,A -85,B 0,C 180,E1 -27696.41,E2 -27696.41} C_VEL
LIN {X 0,Y 238.058,Z 336.677,A -85,B 0,C 180,E1 -27697.682,E2 -27697.682} C_VEL
LIN {X 0,Y 236.618,Z 333.914,A -85,B 0,C 180,E1 -27698.511,E2 -27698.511} C_VEL
LIN {X 0,Y 233.915,Z 332.028,A -85,B 0,C 180,E1 -27699.935,E2 -27699.935} C_VEL
LIN {X 0,Y 232.505,Z 329.7,A -85,B 0,C 180,E1 -27700.819,E2 -27700.819} C_VEL
LIN {X 0,Y 232.135,Z 328.108,A -85,B 0,C 180,E1 -27701.187,E2 -27701.187} C_VEL
LIN {X 0,Y 232.247,Z 328.091,A -85,B 0,C 180,E1 -27706.038,E2 -27706.038} C_VEL
LIN {X 0,Y 232.384,Z 328.073,A -85,B 0,C 180,E1 -27711.332,E2 -27711.332} C_VEL
LIN {X 0,Y 232.569,Z 328.059,A -85,B 0,C 180,E1 -27714.816,E2 -27714.816} C_VEL
LIN {X 0,Y 232.676,Z 328.05,A -85,B 0,C 180,E1 -27718.275,E2 -27718.275} C_VEL
LIN {X 0,Y 232.813,Z 328.032,A -85,B 0,C 180,E1 -27720,E2 -27720} C_VEL
LIN {X 0,Y 232.679,Z 328.043,A -85,B 0,C 180,E1 -27723.452,E2 -27723.452} C_VEL
LIN {X 0,Y 232.529,Z 328.052,A -85,B 0,C 180,E1 -27726.921,E2 -27726.921} C_VEL
LIN {X 0,Y 232.281,Z 328.082,A -85,B 0,C 180,E1 -27732.186,E2 -27732.186} C_VEL
LIN {X 0,Y 232.182,Z 328.11,A -85,B 0,C 180,E1 -27735.754,E2 -27735.754} C_VEL
LIN {X 0,Y 232.139,Z 328.115,A -85,B 0,C 180,E1 -27740.725,E2 -27740.725} C_VEL
LIN {X 0,Y 232.105,Z 328.278,A -85,B 0,C 180,E1 -27744.754,E2 -27744.754} C_VEL
LIN {X 0,Y 233.45,Z 332.46,A -85,B 0,C 180,E1 -27748.69,E2 -27748.69} C_VEL
LIN {X 0,Y 235.043,Z 336.806,A -85,B 0,C 180,E1 -27752.187,E2 -27752.187} C_VEL
LIN {X 0,Y 238.252,Z 341.602,A -85,B 0,C 180,E1 -27753.958,E2 -27753.958} C_VEL
LIN {X 0,Y 240.549,Z 344.456,A -85,B 0,C 180,E1 -27755.106,E2 -27755.106} C_VEL
LIN {X 0,Y 243.779,Z 349.238,A -85,B 0,C 180,E1 -27756.664,E2 -27756.664} C_VEL
LIN {X 0,Y 245.209,Z 351.343,A -85,B 0,C 180,E1 -27757.317,E2 -27757.317} C_VEL
LIN {X 0,Y 249.272,Z 357.639,A -85,B 0,C 180,E1 -27759.086,E2 -27759.086} C_VEL
LIN {X 0,Y 252.867,Z 363.354,A -85,B 0,C 180,E1 -27760.548,E2 -27760.548} C_VEL
LIN {X 0,Y 258.539,Z 372.94,A -85,B 0,C 180,E1 -27762.697,E2 -27762.697} C_VEL
LIN {X 0,Y 265.206,Z 385.382,A -85,B 0,C 180,E1 -27765.034,E2 -27765.034} C_VEL
LIN {X 0,Y 266.209,Z 387.353,A -85,B 0,C 180,E1 -27765.37,E2 -27765.37} C_VEL
LIN {X 0,Y 268.494,Z 393.88,A -85,B 0,C 180,E1 -27766.199,E2 -27766.199} C_VEL
LIN {X 0,Y 270.106,Z 400.999,A -85,B 0,C 180,E1 -27766.867,E2 -27766.867} C_VEL
LIN {X 0,Y 272.167,Z 416.091,A -85,B 0,C 180,E1 -27767.923,E2 -27767.923} C_VEL
LIN {X 0,Y 273.528,Z 430.016,A -85,B 0,C 180,E1 -27768.748,E2 -27768.748} C_VEL
LIN {X 0,Y 270.437,Z 478.847,A -85,B 0,C 180,E1 -27769.955,E2 -27769.955} C_VEL
LIN {X 0,Y 268.548,Z 493.322,A -85,B 0,C 180,E1 -27770.529,E2 -27770.529} C_VEL
LIN {X 0,Y 265.727,Z 507.786,A -85,B 0,C 180,E1 -27771.368,E2 -27771.368} C_VEL
LIN {X 0,Y 262.296,Z 520.654,A -85,B 0,C 180,E1 -27772.354,E2 -27772.354} C_VEL
LIN {X 0,Y 258.351,Z 533.151,A -85,B 0,C 180,E1 -27773.63,E2 -27773.63} C_VEL
LIN {X 0,Y 254.153,Z 544.573,A -85,B 0,C 180,E1 -27775.125,E2 -27775.125} C_VEL
LIN {X 0,Y 249.735,Z 555.091,A -85,B 0,C 180,E1 -27776.849,E2 -27776.849} C_VEL
LIN {X 0,Y 244.943,Z 565.561,A -85,B 0,C 180,E1 -27779.026,E2 -27779.026} C_VEL
LIN {X 0,Y 240.435,Z 574.24,A -85,B 0,C 180,E1 -27781.275,E2 -27781.275} C_VEL
LIN {X 0,Y 235.771,Z 582.608,A -85,B 0,C 180,E1 -27784.016,E2 -27784.016} C_VEL
LIN {X 0,Y 231.713,Z 589.377,A -85,B 0,C 180,E1 -27786.865,E2 -27786.865} C_VEL
LIN {X 0,Y 228.11,Z 595.455,A -85,B 0,C 180,E1 -27790.264,E2 -27790.264} C_VEL
LIN {X 0,Y 225.293,Z 599.983,A -85,B 0,C 180,E1 -27793.756,E2 -27793.756} C_VEL
LIN {X 0,Y 223.318,Z 603.101,A -85,B 0,C 180,E1 -27797.322,E2 -27797.322} C_VEL
LIN {X 0,Y 222.178,Z 604.89,A -85,B 0,C 180,E1 -27800.935,E2 -27800.935} C_VEL
LIN {X 0,Y 221.954,Z 605.391,A -85,B 0,C 180,E1 -27804.572,E2 -27804.572} C_VEL
LIN {X 0,Y 222.565,Z 604.602,A -85,B 0,C 180,E1 -27808.201,E2 -27808.201} C_VEL
LIN {X 0,Y 222.895,Z 604.06,A -85,B 0,C 180,E1 -27809.611,E2 -27809.611} C_VEL
LIN {X 0,Y 222.546,Z 609.338,A -85,B 0,C 180,E1 -27812.71,E2 -27812.71} C_VEL
LIN {X 0,Y 222.33,Z 612.943,A -85,B 0,C 180,E1 -27815.428,E2 -27815.428} C_VEL
LIN {X 0,Y 222.555,Z 616.463,A -85,B 0,C 180,E1 -27819.058,E2 -27819.058} C_VEL
LIN {X 0,Y 223.909,Z 618.719,A -85,B 0,C 180,E1 -27822.653,E2 -27822.653} C_VEL
LIN {X 0,Y 226.311,Z 619.752,A -85,B 0,C 180,E1 -27826.178,E2 -27826.178} C_VEL
LIN {X 0,Y 229.627,Z 619.57,A -85,B 0,C 180,E1 -27829.61,E2 -27829.61} C_VEL
LIN {X 0,Y 233.924,Z 618.179,A -85,B 0,C 180,E1 -27832.913,E2 -27832.913} C_VEL
LIN {X 0,Y 239.278,Z 615.558,A -85,B 0,C 180,E1 -27836.05,E2 -27836.05} C_VEL
LIN {X 0,Y 245.268,Z 611.686,A -85,B 0,C 180,E1 -27839.049,E2 -27839.049} C_VEL
LIN {X 0,Y 252.186,Z 606.431,A -85,B 0,C 180,E1 -27841.856,E2 -27841.856} C_VEL
LIN {X 0,Y 259.963,Z 599.619,A -85,B 0,C 180,E1 -27844.463,E2 -27844.463} C_VEL
LIN {X 0,Y 268.356,Z 591.124,A -85,B 0,C 180,E1 -27846.897,E2 -27846.897} C_VEL
LIN {X 0,Y 276.291,Z 582.05,A -85,B 0,C 180,E1 -27848.866,E2 -27848.866} C_VEL
LIN {X 0,Y 283.496,Z 572.749,A -85,B 0,C 180,E1 -27850.437,E2 -27850.437} C_VEL
LIN {X 0,Y 291.638,Z 560.716,A -85,B 0,C 180,E1 -27852.031,E2 -27852.031} C_VEL
LIN {X 0,Y 298.127,Z 549.754,A -85,B 0,C 180,E1 -27853.158,E2 -27853.158} C_VEL
LIN {X 0,Y 305.022,Z 536.192,A -85,B 0,C 180,E1 -27854.232,E2 -27854.232} C_VEL
LIN {X 0,Y 310.658,Z 523.07,A -85,B 0,C 180,E1 -27855.029,E2 -27855.029} C_VEL
LIN {X 0,Y 316.019,Z 507.57,A -85,B 0,C 180,E1 -27855.745,E2 -27855.745} C_VEL
LIN {X 0,Y 320.342,Z 491.079,A -85,B 0,C 180,E1 -27856.337,E2 -27856.337} C_VEL
LIN {X 0,Y 327.625,Z 455.965,A -85,B 0,C 180,E1 -27857.459,E2 -27857.459} C_VEL
LIN {X 0,Y 327.026,Z 454.192,A -85,B 0,C 180,E1 -27859.424,E2 -27859.424} C_VEL
LIN {X 0,Y 326.728,Z 454.447,A -85,B 0,C 180,E1 -27861.773,E2 -27861.773} C_VEL
LIN {X 0,Y 326.923,Z 456.221,A -85,B 0,C 180,E1 -27863.772,E2 -27863.772} C_VEL
LIN {X 0,Y 327.234,Z 457.791,A -85,B 0,C 180,E1 -27864.862,E2 -27864.862} C_VEL
LIN {X 0,Y 319.022,Z 496.296,A -85,B 0,C 180,E1 -27866.095,E2 -27866.095} C_VEL
LIN {X 0,Y 314.856,Z 510.413,A -85,B 0,C 180,E1 -27866.687,E2 -27866.687} C_VEL
LIN {X 0,Y 309.523,Z 524.864,A -85,B 0,C 180,E1 -27867.492,E2 -27867.492} C_VEL
LIN {X 0,Y 303.766,Z 537.688,A -85,B 0,C 180,E1 -27868.45,E2 -27868.45} C_VEL
LIN {X 0,Y 296.703,Z 550.868,A -85,B 0,C 180,E1 -27869.694,E2 -27869.694} C_VEL
LIN {X 0,Y 289.558,Z 562.272,A -85,B 0,C 180,E1 -27871.066,E2 -27871.066} C_VEL
LIN {X 0,Y 282.163,Z 572.617,A -85,B 0,C 180,E1 -27872.661,E2 -27872.661} C_VEL
LIN {X 0,Y 273.861,Z 582.632,A -85,B 0,C 180,E1 -27874.633,E2 -27874.633} C_VEL
LIN {X 0,Y 266.156,Z 590.769,A -85,B 0,C 180,E1 -27876.749,E2 -27876.749} C_VEL
LIN {X 0,Y 259.977,Z 596.554,A -85,B 0,C 180,E1 -27878.671,E2 -27878.671} C_VEL
LIN {X 0,Y 252.335,Z 602.745,A -85,B 0,C 180,E1 -27881.384,E2 -27881.384} C_VEL
LIN {X 0,Y 247.103,Z 606.405,A -85,B 0,C 180,E1 -27883.533,E2 -27883.533} C_VEL
LIN {X 0,Y 240.713,Z 609.998,A -85,B 0,C 180,E1 -27886.539,E2 -27886.539} C_VEL
LIN {X 0,Y 235.201,Z 612.238,A -85,B 0,C 180,E1 -27889.707,E2 -27889.707} C_VEL
LIN {X 0,Y 230.704,Z 613.18,A -85,B 0,C 180,E1 -27893.024,E2 -27893.024} C_VEL
LIN {X 0,Y 227.129,Z 612.862,A -85,B 0,C 180,E1 -27896.464,E2 -27896.464} C_VEL
LIN {X 0,Y 224.632,Z 611.294,A -85,B 0,C 180,E1 -27900,E2 -27900} C_VEL
LIN {X 0,Y 222.957,Z 608.436,A -85,B 0,C 180,E1 -27903.602,E2 -27903.602} C_VEL
LIN {X 0,Y 222.027,Z 604.197,A -85,B 0,C 180,E1 -27907.249,E2 -27907.249} C_VEL
LIN {X 0,Y 221.911,Z 598.451,A -85,B 0,C 180,E1 -27910.917,E2 -27910.917} C_VEL
LIN {X 0,Y 222.046,Z 591.877,A -85,B 0,C 180,E1 -27914.151,E2 -27914.151} C_VEL
LIN {X 0,Y 222.372,Z 584.896,A -85,B 0,C 180,E1 -27916.94,E2 -27916.94} C_VEL
LIN {X 0,Y 222.814,Z 576.709,A -85,B 0,C 180,E1 -27919.649,E2 -27919.649} C_VEL
LIN {X 0,Y 223.364,Z 567.823,A -85,B 0,C 180,E1 -27922.105,E2 -27922.105} C_VEL
LIN {X 0,Y 224.172,Z 557.183,A -85,B 0,C 180,E1 -27924.573,E2 -27924.573} C_VEL
LIN {X 0,Y 225.123,Z 545.53,A -85,B 0,C 180,E1 -27926.817,E2 -27926.817} C_VEL
LIN {X 0,Y 226.132,Z 533.729,A -85,B 0,C 180,E1 -27928.693,E2 -27928.693} C_VEL
LIN {X 0,Y 227.338,Z 519.354,A -85,B 0,C 180,E1 -27930.525,E2 -27930.525} C_VEL
LIN {X 0,Y 228.362,Z 505.151,A -85,B 0,C 180,E1 -27931.945,E2 -27931.945} C_VEL
LIN {X 0,Y 229.355,Z 489.841,A -85,B 0,C 180,E1 -27933.086,E2 -27933.086} C_VEL
LIN {X 0,Y 230.914,Z 455.17,A -85,B 0,C 180,E1 -27934.867,E2 -27934.867} C_VEL
LIN {X 0,Y 233.907,Z 391.367,A -85,B 0,C 180,E1 -27937.975,E2 -27937.975} C_VEL
LIN {X 0,Y 231.423,Z 364.275,A -85,B 0,C 180,E1 -27939.407,E2 -27939.407} C_VEL
LIN {X 0,Y 230.8,Z 356.13,A -85,B 0,C 180,E1 -27939.839,E2 -27939.839} C_VEL
LIN {X 0,Y 228.739,Z 347.522,A -85,B 0,C 180,E1 -27940.378,E2 -27940.378} C_VEL
LIN {X 0,Y 225.292,Z 330.321,A -85,B 0,C 180,E1 -27944.752,E2 -27944.752} C_VEL
LIN {X 0,Y 225.018,Z 329.003,A -85,B 0,C 180,E1 -27945.137,E2 -27945.137} C_VEL
LIN {X 0,Y 224.965,Z 329.017,A -85,B 0,C 180,E1 -27949.163,E2 -27949.163} C_VEL
LIN {X 0,Y 224.931,Z 329.018,A -85,B 0,C 180,E1 -27953.72,E2 -27953.72} C_VEL
LIN {X 0,Y 224.951,Z 329.015,A -85,B 0,C 180,E1 -27958.035,E2 -27958.035} C_VEL
LIN {X 0,Y 224.984,Z 329.001,A -85,B 0,C 180,E1 -27962.156,E2 -27962.156} C_VEL
LIN {X 0,Y 225.032,Z 329.013,A -85,B 0,C 180,E1 -27964.675,E2 -27964.675} C_VEL
LIN {X 0,Y 226.112,Z 331.977,A -85,B 0,C 180,E1 -27964.976,E2 -27964.976} C_VEL
LIN {X 0,Y 227.721,Z 334.641,A -85,B 0,C 180,E1 -27965.33,E2 -27965.33} C_VEL
LIN {X 0,Y 236.598,Z 351.282,A -85,B 0,C 180,E1 -27967.243,E2 -27967.243} C_VEL
LIN {X 0,Y 244.25,Z 368.44,A -85,B 0,C 180,E1 -27968.848,E2 -27968.848} C_VEL
LIN {X 0,Y 245.57,Z 371.672,A -85,B 0,C 180,E1 -27969.122,E2 -27969.122} C_VEL
LIN {X 0,Y 242.271,Z 455.232,A -85,B 0,C 180,E1 -27971.507,E2 -27971.507} C_VEL
LIN {X 0,Y 241.232,Z 468.9,A -85,B 0,C 180,E1 -27972.191,E2 -27972.191} C_VEL
LIN {X 0,Y 239.8,Z 482.902,A -85,B 0,C 180,E1 -27973.231,E2 -27973.231} C_VEL
LIN {X 0,Y 237.967,Z 496.766,A -85,B 0,C 180,E1 -27974.634,E2 -27974.634} C_VEL
LIN {X 0,Y 235.674,Z 509.264,A -85,B 0,C 180,E1 -27976.241,E2 -27976.241} C_VEL
LIN {X 0,Y 233.349,Z 520.664,A -85,B 0,C 180,E1 -27978.086,E2 -27978.086} C_VEL
LIN {X 0,Y 231.461,Z 530.119,A -85,B 0,C 180,E1 -27979.975,E2 -27979.975} C_VEL
LIN {X 0,Y 228.97,Z 540.699,A -85,B 0,C 180,E1 -27982.526,E2 -27982.526} C_VEL
LIN {X 0,Y 227.015,Z 549.412,A -85,B 0,C 180,E1 -27985.128,E2 -27985.128} C_VEL
LIN {X 0,Y 225.267,Z 556.686,A -85,B 0,C 180,E1 -27987.768,E2 -27987.768} C_VEL
LIN {X 0,Y 224.162,Z 563.343,A -85,B 0,C 180,E1 -27990.76,E2 -27990.76} C_VEL
LIN {X 0,Y 223.227,Z 568.442,A -85,B 0,C 180,E1 -27993.594,E2 -27993.594} C_VEL
LIN {X 0,Y 222.309,Z 573.477,A -85,B 0,C 180,E1 -27997.236,E2 -27997.236} C_VEL
LIN {X 0,Y 222.104,Z 577.006,A -85,B 0,C 180,E1 -28000.903,E2 -28000.903} C_VEL
LIN {X 0,Y 222.296,Z 579.151,A -85,B 0,C 180,E1 -28004.596,E2 -28004.596} C_VEL
LIN {X 0,Y 223.137,Z 579.927,A -85,B 0,C 180,E1 -28008.29,E2 -28008.29} C_VEL
LIN {X 0,Y 224.577,Z 579.326,A -85,B 0,C 180,E1 -28011.974,E2 -28011.974} C_VEL
LIN {X 0,Y 226.75,Z 577.33,A -85,B 0,C 180,E1 -28015.619,E2 -28015.619} C_VEL
LIN {X 0,Y 229.679,Z 573.88,A -85,B 0,C 180,E1 -28019.2,E2 -28019.2} C_VEL
LIN {X 0,Y 233.342,Z 568.862,A -85,B 0,C 180,E1 -28022.7,E2 -28022.7} C_VEL
LIN {X 0,Y 236.647,Z 563.942,A -85,B 0,C 180,E1 -28025.246,E2 -28025.246} C_VEL
LIN {X 0,Y 241.059,Z 556.652,A -85,B 0,C 180,E1 -28028.192,E2 -28028.192} C_VEL
LIN {X 0,Y 245.099,Z 549.25,A -85,B 0,C 180,E1 -28030.547,E2 -28030.547} C_VEL
LIN {X 0,Y 249.634,Z 540.156,A -85,B 0,C 180,E1 -28032.858,E2 -28032.858} C_VEL
LIN {X 0,Y 254.57,Z 528.973,A -85,B 0,C 180,E1 -28035.107,E2 -28035.107} C_VEL
LIN {X 0,Y 258.901,Z 517.523,A -85,B 0,C 180,E1 -28036.92,E2 -28036.92} C_VEL
LIN {X 0,Y 262.953,Z 504.73,A -85,B 0,C 180,E1 -28038.513,E2 -28038.513} C_VEL
LIN {X 0,Y 266.385,Z 491.203,A -85,B 0,C 180,E1 -28039.827,E2 -28039.827} C_VEL
LIN {X 0,Y 268.943,Z 478.279,A -85,B 0,C 180,E1 -28040.782,E2 -28040.782} C_VEL
LIN {X 0,Y 270.948,Z 464.311,A -85,B 0,C 180,E1 -28041.534,E2 -28041.534} C_VEL
LIN {X 0,Y 272.308,Z 449.821,A -85,B 0,C 180,E1 -28042.024,E2 -28042.024} C_VEL
LIN {X 0,Y 275.106,Z 402.332,A -85,B 0,C 180,E1 -28043.193,E2 -28043.193} C_VEL
LIN {X 0,Y 271.575,Z 395.186,A -85,B 0,C 180,E1 -28044.267,E2 -28044.267} C_VEL
LIN {X 0,Y 264.963,Z 383.525,A -85,B 0,C 180,E1 -28046.356,E2 -28046.356} C_VEL
LIN {X 0,Y 257.408,Z 371.419,A -85,B 0,C 180,E1 -28048.946,E2 -28048.946} C_VEL
LIN {X 0,Y 250.94,Z 362.226,A -85,B 0,C 180,E1 -28051.38,E2 -28051.38} C_VEL
LIN {X 0,Y 247.652,Z 357.775,A -85,B 0,C 180,E1 -28052.717,E2 -28052.717} C_VEL
LIN {X 0,Y 245.244,Z 354.477,A -85,B 0,C 180,E1 -28053.752,E2 -28053.752} C_VEL
LIN {X 0,Y 241.908,Z 350.118,A -85,B 0,C 180,E1 -28055.264,E2 -28055.264} C_VEL
LIN {X 0,Y 239.047,Z 346.502,A -85,B 0,C 180,E1 -28056.648,E2 -28056.648} C_VEL
LIN {X 0,Y 238.171,Z 345.339,A -85,B 0,C 180,E1 -28057.094,E2 -28057.094} C_VEL
LIN {X 0,Y 235.48,Z 342.44,A -85,B 0,C 180,E1 -28058.488,E2 -28058.488} C_VEL
LIN {X 0,Y 234.345,Z 340.389,A -85,B 0,C 180,E1 -28059.16,E2 -28059.16} C_VEL
LIN {X 0,Y 231.539,Z 337.97,A -85,B 0,C 180,E1 -28060.735,E2 -28060.735} C_VEL
LIN {X 0,Y 229.789,Z 334.832,A -85,B 0,C 180,E1 -28061.909,E2 -28061.909} C_VEL
LIN {X 0,Y 227.19,Z 333.227,A -85,B 0,C 180,E1 -28063.545,E2 -28063.545} C_VEL
LIN {X 0,Y 225.729,Z 331,A -85,B 0,C 180,E1 -28064.65,E2 -28064.65} C_VEL
LIN {X 0,Y 225.191,Z 328.972,A -85,B 0,C 180,E1 -28065.245,E2 -28065.245} C_VEL
LIN {X 0,Y 225.25,Z 328.975,A -85,B 0,C 180,E1 -28069.247,E2 -28069.247} C_VEL
LIN {X 0,Y 225.57,Z 328.945,A -85,B 0,C 180,E1 -28073.504,E2 -28073.504} C_VEL
LIN {X 0,Y 225.64,Z 328.925,A -85,B 0,C 180,E1 -28078.221,E2 -28078.221} C_VEL
LIN {X 0,Y 225.764,Z 328.909,A -85,B 0,C 180,E1 -28080,E2 -28080} C_VEL
LIN {X 0,Y 225.625,Z 328.923,A -85,B 0,C 180,E1 -28083.56,E2 -28083.56} C_VEL
LIN {X 0,Y 225.47,Z 328.93,A -85,B 0,C 180,E1 -28087.138,E2 -28087.138} C_VEL
LIN {X 0,Y 225.214,Z 328.961,A -85,B 0,C 180,E1 -28092.575,E2 -28092.575} C_VEL
LIN {X 0,Y 225.093,Z 328.985,A -85,B 0,C 180,E1 -28096.264,E2 -28096.264} C_VEL
LIN {X 0,Y 225.072,Z 329.017,A -85,B 0,C 180,E1 -28101.007,E2 -28101.007} C_VEL
LIN {X 0,Y 226.673,Z 333.901,A -85,B 0,C 180,E1 -28106.358,E2 -28106.358} C_VEL
LIN {X 0,Y 227.445,Z 335.834,A -85,B 0,C 180,E1 -28108.074,E2 -28108.074} C_VEL
LIN {X 0,Y 230.386,Z 340.292,A -85,B 0,C 180,E1 -28110.078,E2 -28110.078} C_VEL
LIN {X 0,Y 233.137,Z 343.576,A -85,B 0,C 180,E1 -28111.721,E2 -28111.721} C_VEL
LIN {X 0,Y 236.148,Z 348.016,A -85,B 0,C 180,E1 -28113.428,E2 -28113.428} C_VEL
LIN {X 0,Y 238.053,Z 350.518,A -85,B 0,C 180,E1 -28114.421,E2 -28114.421} C_VEL
LIN {X 0,Y 241.538,Z 355.618,A -85,B 0,C 180,E1 -28116.154,E2 -28116.154} C_VEL
LIN {X 0,Y 246.602,Z 363.752,A -85,B 0,C 180,E1 -28118.477,E2 -28118.477} C_VEL
LIN {X 0,Y 249.98,Z 369.258,A -85,B 0,C 180,E1 -28119.904,E2 -28119.904} C_VEL
LIN {X 0,Y 255.159,Z 378.256,A -85,B 0,C 180,E1 -28121.955,E2 -28121.955} C_VEL
LIN {X 0,Y 262.098,Z 391.472,A -85,B 0,C 180,E1 -28124.482,E2 -28124.482} C_VEL
LIN {X 0,Y 268.434,Z 405.348,A -85,B 0,C 180,E1 -28126.642,E2 -28126.642} C_VEL
LIN {X 0,Y 271.984,Z 414.654,A -85,B 0,C 180,E1 -28127.828,E2 -28127.828} C_VEL
LIN {X 0,Y 272.167,Z 416.091,A -85,B 0,C 180,E1 -28127.923,E2 -28127.923} C_VEL
LIN {X 0,Y 272.315,Z 419.929,A -85,B 0,C 180,E1 -28128.102,E2 -28128.102} C_VEL
LIN {X 0,Y 272.006,Z 423.845,A -85,B 0,C 180,E1 -28128.182,E2 -28128.182} C_VEL
LIN {X 0,Y 270.542,Z 431.683,A -85,B 0,C 180,E1 -28128.154,E2 -28128.154} C_VEL
LIN {X 0,Y 268.023,Z 443.583,A -85,B 0,C 180,E1 -28128.044,E2 -28128.044} C_VEL
LIN {X 0,Y 267.604,Z 447.59,A -85,B 0,C 180,E1 -28128.104,E2 -28128.104} C_VEL
LIN {X 0,Y 265.358,Z 479.442,A -85,B 0,C 180,E1 -28128.902,E2 -28128.902} C_VEL
LIN {X 0,Y 263.41,Z 493.582,A -85,B 0,C 180,E1 -28129.477,E2 -28129.477} C_VEL
LIN {X 0,Y 260.796,Z 506.746,A -85,B 0,C 180,E1 -28130.247,E2 -28130.247} C_VEL
LIN {X 0,Y 257.276,Z 519.748,A -85,B 0,C 180,E1 -28131.236,E2 -28131.236} C_VEL
LIN {X 0,Y 253.194,Z 532.341,A -85,B 0,C 180,E1 -28132.516,E2 -28132.516} C_VEL
LIN {X 0,Y 248.867,Z 543.832,A -85,B 0,C 180,E1 -28134.023,E2 -28134.023} C_VEL
LIN {X 0,Y 244.707,Z 553.433,A -85,B 0,C 180,E1 -28135.581,E2 -28135.581} C_VEL
LIN {X 0,Y 239.704,Z 564.107,A -85,B 0,C 180,E1 -28137.778,E2 -28137.778} C_VEL
LIN {X 0,Y 234.987,Z 572.957,A -85,B 0,C 180,E1 -28140.053,E2 -28140.053} C_VEL
LIN {X 0,Y 230.011,Z 581.475,A -85,B 0,C 180,E1 -28142.825,E2 -28142.825} C_VEL
LIN {X 0,Y 226.342,Z 587.468,A -85,B 0,C 180,E1 -28145.311,E2 -28145.311} C_VEL
LIN {X 0,Y 222.265,Z 593.908,A -85,B 0,C 180,E1 -28148.757,E2 -28148.757} C_VEL
LIN {X 0,Y 219.11,Z 598.766,A -85,B 0,C 180,E1 -28152.325,E2 -28152.325} C_VEL
LIN {X 0,Y 216.974,Z 601.847,A -85,B 0,C 180,E1 -28155.574,E2 -28155.574} C_VEL
LIN {X 0,Y 215.62,Z 603.812,A -85,B 0,C 180,E1 -28158.765,E2 -28158.765} C_VEL
LIN {X 0,Y 214.842,Z 604.896,A -85,B 0,C 180,E1 -28162.511,E2 -28162.511} C_VEL
LIN {X 0,Y 215.085,Z 604.703,A -85,B 0,C 180,E1 -28166.27,E2 -28166.27} C_VEL
LIN {X 0,Y 215.92,Z 603.256,A -85,B 0,C 180,E1 -28170.005,E2 -28170.005} C_VEL
LIN {X 0,Y 215.591,Z 608.015,A -85,B 0,C 180,E1 -28172.798,E2 -28172.798} C_VEL
LIN {X 0,Y 215.336,Z 612.872,A -85,B 0,C 180,E1 -28176.542,E2 -28176.542} C_VEL
LIN {X 0,Y 215.591,Z 615.549,A -85,B 0,C 180,E1 -28179.353,E2 -28179.353} C_VEL
LIN {X 0,Y 217.003,Z 618.072,A -85,B 0,C 180,E1 -28183.063,E2 -28183.063} C_VEL
LIN {X 0,Y 219.848,Z 619.462,A -85,B 0,C 180,E1 -28187.096,E2 -28187.096} C_VEL
LIN {X 0,Y 222.95,Z 619.489,A -85,B 0,C 180,E1 -28190.222,E2 -28190.222} C_VEL
LIN {X 0,Y 227.416,Z 618.408,A -85,B 0,C 180,E1 -28193.608,E2 -28193.608} C_VEL
LIN {X 0,Y 232.96,Z 616.114,A -85,B 0,C 180,E1 -28196.813,E2 -28196.813} C_VEL
LIN {X 0,Y 239.145,Z 612.592,A -85,B 0,C 180,E1 -28199.867,E2 -28199.867} C_VEL
LIN {X 0,Y 246.294,Z 607.722,A -85,B 0,C 180,E1 -28202.711,E2 -28202.711} C_VEL
LIN {X 0,Y 254.291,Z 601.392,A -85,B 0,C 180,E1 -28205.345,E2 -28205.345} C_VEL
LIN {X 0,Y 262.91,Z 593.476,A -85,B 0,C 180,E1 -28207.794,E2 -28207.794} C_VEL
LIN {X 0,Y 271.045,Z 584.947,A -85,B 0,C 180,E1 -28209.766,E2 -28209.766} C_VEL
LIN {X 0,Y 279.656,Z 574.598,A -85,B 0,C 180,E1 -28211.589,E2 -28211.589} C_VEL
LIN {X 0,Y 287.36,Z 564.027,A -85,B 0,C 180,E1 -28213.043,E2 -28213.043} C_VEL
LIN {X 0,Y 294.81,Z 552.354,A -85,B 0,C 180,E1 -28214.289,E2 -28214.289} C_VEL
LIN {X 0,Y 301.701,Z 539.817,A -85,B 0,C 180,E1 -28215.32,E2 -28215.32} C_VEL
LIN {X 0,Y 308.175,Z 525.835,A -85,B 0,C 180,E1 -28216.194,E2 -28216.194} C_VEL
LIN {X 0,Y 314.067,Z 510.101,A -85,B 0,C 180,E1 -28216.924,E2 -28216.924} C_VEL
LIN {X 0,Y 318.323,Z 495.356,A -85,B 0,C 180,E1 -28217.469,E2 -28217.469} C_VEL
LIN {X 0,Y 325.586,Z 461.981,A -85,B 0,C 180,E1 -28218.507,E2 -28218.507} C_VEL
LIN {X 0,Y 325.329,Z 461.041,A -85,B 0,C 180,E1 -28219.766,E2 -28219.766} C_VEL
LIN {X 0,Y 325.122,Z 461.391,A -85,B 0,C 180,E1 -28221.765,E2 -28221.765} C_VEL
LIN {X 0,Y 325.288,Z 463.173,A -85,B 0,C 180,E1 -28223.711,E2 -28223.711} C_VEL
LIN {X 0,Y 325.299,Z 463.274,A -85,B 0,C 180,E1 -28223.787,E2 -28223.787} C_VEL
LIN {X 0,Y 317.947,Z 496.519,A -85,B 0,C 180,E1 -28224.825,E2 -28224.825} C_VEL
LIN {X 0,Y 313.691,Z 510.504,A -85,B 0,C 180,E1 -28225.389,E2 -28225.389} C_VEL
LIN {X 0,Y 308.202,Z 524.943,A -85,B 0,C 180,E1 -28226.165,E2 -28226.165} C_VEL
LIN {X 0,Y 302.629,Z 537.022,A -85,B 0,C 180,E1 -28227.035,E2 -28227.035} C_VEL
LIN {X 0,Y 296.155,Z 548.945,A -85,B 0,C 180,E1 -28228.087,E2 -28228.087} C_VEL
LIN {X 0,Y 288.848,Z 560.444,A -85,B 0,C 180,E1 -28229.387,E2 -28229.387} C_VEL
LIN {X 0,Y 281.829,Z 570.133,A -85,B 0,C 180,E1 -28230.761,E2 -28230.761} C_VEL
LIN {X 0,Y 273.598,Z 580.056,A -85,B 0,C 180,E1 -28232.56,E2 -28232.56} C_VEL
LIN {X 0,Y 265.303,Z 588.741,A -85,B 0,C 180,E1 -28234.594,E2 -28234.594} C_VEL
LIN {X 0,Y 257.59,Z 595.794,A -85,B 0,C 180,E1 -28236.778,E2 -28236.778} C_VEL
LIN {X 0,Y 249.443,Z 602.206,A -85,B 0,C 180,E1 -28239.451,E2 -28239.451} C_VEL
LIN {X 0,Y 243.5,Z 606.145,A -85,B 0,C 180,E1 -28241.681,E2 -28241.681} C_VEL
LIN {X 0,Y 236.898,Z 609.758,A -85,B 0,C 180,E1 -28244.567,E2 -28244.567} C_VEL
LIN {X 0,Y 230.836,Z 612.194,A -85,B 0,C 180,E1 -28247.736,E2 -28247.736} C_VEL
LIN {X 0,Y 225.755,Z 613.331,A -85,B 0,C 180,E1 -28251.075,E2 -28251.075} C_VEL
LIN {X 0,Y 221.614,Z 613.209,A -85,B 0,C 180,E1 -28254.559,E2 -28254.559} C_VEL
LIN {X 0,Y 218.589,Z 611.844,A -85,B 0,C 180,E1 -28258.164,E2 -28258.164} C_VEL
LIN {X 0,Y 216.562,Z 609.235,A -85,B 0,C 180,E1 -28261.853,E2 -28261.853} C_VEL
LIN {X 0,Y 215.294,Z 605.284,A -85,B 0,C 180,E1 -28265.601,E2 -28265.601} C_VEL
LIN {X 0,Y 214.897,Z 599.863,A -85,B 0,C 180,E1 -28269.379,E2 -28269.379} C_VEL
LIN {X 0,Y 214.916,Z 594.296,A -85,B 0,C 180,E1 -28272.417,E2 -28272.417} C_VEL
LIN {X 0,Y 215.237,Z 587.164,A -85,B 0,C 180,E1 -28275.574,E2 -28275.574} C_VEL
LIN {X 0,Y 215.64,Z 579.147,A -85,B 0,C 180,E1 -28278.463,E2 -28278.463} C_VEL
LIN {X 0,Y 216.204,Z 569.34,A -85,B 0,C 180,E1 -28281.375,E2 -28281.375} C_VEL
LIN {X 0,Y 216.964,Z 558.421,A -85,B 0,C 180,E1 -28284.053,E2 -28284.053} C_VEL
LIN {X 0,Y 217.95,Z 546.075,A -85,B 0,C 180,E1 -28286.539,E2 -28286.539} C_VEL
LIN {X 0,Y 219.059,Z 533.138,A -85,B 0,C 180,E1 -28288.661,E2 -28288.661} C_VEL
LIN {X 0,Y 220.29,Z 518.449,A -85,B 0,C 180,E1 -28290.58,E2 -28290.58} C_VEL
LIN {X 0,Y 221.3,Z 504.624,A -85,B 0,C 180,E1 -28291.995,E2 -28291.995} C_VEL
LIN {X 0,Y 222.252,Z 489.733,A -85,B 0,C 180,E1 -28293.134,E2 -28293.134} C_VEL
LIN {X 0,Y 223.486,Z 461.963,A -85,B 0,C 180,E1 -28294.622,E2 -28294.622} C_VEL
LIN {X 0,Y 226.834,Z 391.544,A -85,B 0,C 180,E1 -28298.193,E2 -28298.193} C_VEL
LIN {X 0,Y 224.402,Z 364.457,A -85,B 0,C 180,E1 -28299.677,E2 -28299.677} C_VEL
LIN {X 0,Y 223.797,Z 357.272,A -85,B 0,C 180,E1 -28300.074,E2 -28300.074} C_VEL
LIN {X 0,Y 221.497,Z 347.448,A -85,B 0,C 180,E1 -28300.734,E2 -28300.734} C_VEL
LIN {X 0,Y 217.973,Z 329.88,A -85,B 0,C 180,E1 -28305.331,E2 -28305.331} C_VEL
LIN {X 0,Y 217.914,Z 329.892,A -85,B 0,C 180,E1 -28310.483,E2 -28310.483} C_VEL
LIN {X 0,Y 217.879,Z 329.886,A -85,B 0,C 180,E1 -28314.638,E2 -28314.638} C_VEL
LIN {X 0,Y 217.904,Z 329.9,A -85,B 0,C 180,E1 -28319.044,E2 -28319.044} C_VEL
LIN {X 0,Y 217.918,Z 329.897,A -85,B 0,C 180,E1 -28323.519,E2 -28323.519} C_VEL
LIN {X 0,Y 218.987,Z 332.811,A -85,B 0,C 180,E1 -28323.819,E2 -28323.819} C_VEL
LIN {X 0,Y 220.666,Z 335.538,A -85,B 0,C 180,E1 -28324.212,E2 -28324.212} C_VEL
LIN {X 0,Y 228.252,Z 349.222,A -85,B 0,C 180,E1 -28325.946,E2 -28325.946} C_VEL
LIN {X 0,Y 235.098,Z 363.551,A -85,B 0,C 180,E1 -28327.459,E2 -28327.459} C_VEL
LIN {X 0,Y 239.308,Z 373.55,A -85,B 0,C 180,E1 -28328.377,E2 -28328.377} C_VEL
LIN {X 0,Y 235.959,Z 454.707,A -85,B 0,C 180,E1 -28330.73,E2 -28330.73} C_VEL
LIN {X 0,Y 234.839,Z 469.243,A -85,B 0,C 180,E1 -28331.464,E2 -28331.464} C_VEL
LIN {X 0,Y 233.35,Z 483.263,A -85,B 0,C 180,E1 -28332.528,E2 -28332.528} C_VEL
LIN {X 0,Y 231.456,Z 497.134,A -85,B 0,C 180,E1 -28333.966,E2 -28333.966} C_VEL
LIN {X 0,Y 229.067,Z 509.646,A -85,B 0,C 180,E1 -28335.61,E2 -28335.61} C_VEL
LIN {X 0,Y 226.659,Z 521.052,A -85,B 0,C 180,E1 -28337.503,E2 -28337.503} C_VEL
LIN {X 0,Y 224.504,Z 531.478,A -85,B 0,C 180,E1 -28339.661,E2 -28339.661} C_VEL
LIN {X 0,Y 221.922,Z 541.909,A -85,B 0,C 180,E1 -28342.287,E2 -28342.287} C_VEL
LIN {X 0,Y 219.949,Z 550.487,A -85,B 0,C 180,E1 -28344.971,E2 -28344.971} C_VEL
LIN {X 0,Y 218.187,Z 557.644,A -85,B 0,C 180,E1 -28347.696,E2 -28347.696} C_VEL
LIN {X 0,Y 217.008,Z 564.464,A -85,B 0,C 180,E1 -28350.919,E2 -28350.919} C_VEL
LIN {X 0,Y 216.08,Z 569.21,A -85,B 0,C 180,E1 -28353.713,E2 -28353.713} C_VEL
LIN {X 0,Y 215.177,Z 574.159,A -85,B 0,C 180,E1 -28357.477,E2 -28357.477} C_VEL
LIN {X 0,Y 215.042,Z 577.604,A -85,B 0,C 180,E1 -28361.265,E2 -28361.265} C_VEL
LIN {X 0,Y 215.265,Z 579.663,A -85,B 0,C 180,E1 -28365.084,E2 -28365.084} C_VEL
LIN {X 0,Y 216.212,Z 580.338,A -85,B 0,C 180,E1 -28368.898,E2 -28368.898} C_VEL
LIN {X 0,Y 217.803,Z 579.65,A -85,B 0,C 180,E1 -28372.695,E2 -28372.695} C_VEL
LIN {X 0,Y 220.163,Z 577.573,A -85,B 0,C 180,E1 -28376.444,E2 -28376.444} C_VEL
LIN {X 0,Y 223.291,Z 574.038,A -85,B 0,C 180,E1 -28380.12,E2 -28380.12} C_VEL
LIN {X 0,Y 227.204,Z 568.929,A -85,B 0,C 180,E1 -28383.699,E2 -28383.699} C_VEL
LIN {X 0,Y 230.716,Z 563.912,A -85,B 0,C 180,E1 -28386.294,E2 -28386.294} C_VEL
LIN {X 0,Y 235.357,Z 556.49,A -85,B 0,C 180,E1 -28389.305,E2 -28389.305} C_VEL
LIN {X 0,Y 239.584,Z 548.993,A -85,B 0,C 180,E1 -28391.685,E2 -28391.685} C_VEL
LIN {X 0,Y 244.662,Z 539.073,A -85,B 0,C 180,E1 -28394.184,E2 -28394.184} C_VEL
LIN {X 0,Y 249.448,Z 528.354,A -85,B 0,C 180,E1 -28396.3,E2 -28396.3} C_VEL
LIN {X 0,Y 253.956,Z 516.645,A -85,B 0,C 180,E1 -28398.126,E2 -28398.126} C_VEL
LIN {X 0,Y 257.683,Z 505.179,A -85,B 0,C 180,E1 -28399.555,E2 -28399.555} C_VEL
LIN {X 0,Y 261.233,Z 491.662,A -85,B 0,C 180,E1 -28400.88,E2 -28400.88} C_VEL
LIN {X 0,Y 263.872,Z 478.756,A -85,B 0,C 180,E1 -28401.842,E2 -28401.842} C_VEL
LIN {X 0,Y 265.932,Z 464.922,A -85,B 0,C 180,E1 -28402.595,E2 -28402.595} C_VEL
LIN {X 0,Y 267.368,Z 450.147,A -85,B 0,C 180,E1 -28403.1,E2 -28403.1} C_VEL
LIN {X 0,Y 270.125,Z 404.938,A -85,B 0,C 180,E1 -28404.225,E2 -28404.225} C_VEL
LIN {X 0,Y 264.681,Z 394.398,A -85,B 0,C 180,E1 -28405.976,E2 -28405.976} C_VEL
LIN {X 0,Y 257.579,Z 382.352,A -85,B 0,C 180,E1 -28408.404,E2 -28408.404} C_VEL
LIN {X 0,Y 251.616,Z 373.09,A -85,B 0,C 180,E1 -28410.63,E2 -28410.63} C_VEL
LIN {X 0,Y 245.453,Z 364.383,A -85,B 0,C 180,E1 -28413.148,E2 -28413.148} C_VEL
LIN {X 0,Y 242.183,Z 359.985,A -85,B 0,C 180,E1 -28414.599,E2 -28414.599} C_VEL
LIN {X 0,Y 239.445,Z 356.239,A -85,B 0,C 180,E1 -28415.903,E2 -28415.903} C_VEL
LIN {X 0,Y 236.439,Z 352.26,A -85,B 0,C 180,E1 -28417.429,E2 -28417.429} C_VEL
LIN {X 0,Y 233.048,Z 348.316,A -85,B 0,C 180,E1 -28419.259,E2 -28419.259} C_VEL
LIN {X 0,Y 232.007,Z 346.706,A -85,B 0,C 180,E1 -28419.884,E2 -28419.884} C_VEL
LIN {X 0,Y 229.213,Z 343.885,A -85,B 0,C 180,E1 -28421.552,E2 -28421.552} C_VEL
LIN {X 0,Y 227.926,Z 341.539,A -85,B 0,C 180,E1 -28422.452,E2 -28422.452} C_VEL
LIN {X 0,Y 225.222,Z 339.499,A -85,B 0,C 180,E1 -28424.251,E2 -28424.251} C_VEL
LIN {X 0,Y 223.621,Z 336.797,A -85,B 0,C 180,E1 -28425.546,E2 -28425.546} C_VEL
LIN {X 0,Y 223.21,Z 335.789,A -85,B 0,C 180,E1 -28425.925,E2 -28425.925} C_VEL
LIN {X 0,Y 220.408,Z 334.234,A -85,B 0,C 180,E1 -28428.195,E2 -28428.195} C_VEL
LIN {X 0,Y 218.731,Z 331.753,A -85,B 0,C 180,E1 -28429.914,E2 -28429.914} C_VEL
LIN {X 0,Y 218.247,Z 329.833,A -85,B 0,C 180,E1 -28430.649,E2 -28430.649} C_VEL
LIN {X 0,Y 218.537,Z 329.82,A -85,B 0,C 180,E1 -28433.465,E2 -28433.465} C_VEL
LIN {X 0,Y 218.604,Z 329.8,A -85,B 0,C 180,E1 -28438.164,E2 -28438.164} C_VEL
LIN {X 0,Y 218.718,Z 329.786,A -85,B 0,C 180,E1 -28440,E2 -28440} C_VEL
LIN {X 0,Y 218.574,Z 329.802,A -85,B 0,C 180,E1 -28443.675,E2 -28443.675} C_VEL
LIN {X 0,Y 218.413,Z 329.808,A -85,B 0,C 180,E1 -28447.37,E2 -28447.37} C_VEL
LIN {X 0,Y 218.207,Z 329.843,A -85,B 0,C 180,E1 -28451.105,E2 -28451.105} C_VEL
LIN {X 0,Y 218.084,Z 329.86,A -85,B 0,C 180,E1 -28456.049,E2 -28456.049} C_VEL
LIN {X 0,Y 219.087,Z 332.77,A -85,B 0,C 180,E1 -28460.59,E2 -28460.59} C_VEL
LIN {X 0,Y 219.532,Z 334.356,A -85,B 0,C 180,E1 -28462.336,E2 -28462.336} C_VEL
LIN {X 0,Y 224.242,Z 340.814,A -85,B 0,C 180,E1 -28466.482,E2 -28466.482} C_VEL
LIN {X 0,Y 225.578,Z 342.34,A -85,B 0,C 180,E1 -28467.464,E2 -28467.464} C_VEL
LIN {X 0,Y 229.597,Z 348.117,A -85,B 0,C 180,E1 -28470.224,E2 -28470.224} C_VEL
LIN {X 0,Y 231.008,Z 349.937,A -85,B 0,C 180,E1 -28471.092,E2 -28471.092} C_VEL
LIN {X 0,Y 234.683,Z 355.2,A -85,B 0,C 180,E1 -28473.222,E2 -28473.222} C_VEL
LIN {X 0,Y 239.78,Z 362.985,A -85,B 0,C 180,E1 -28475.878,E2 -28475.878} C_VEL
LIN {X 0,Y 244.067,Z 370.046,A -85,B 0,C 180,E1 -28477.904,E2 -28477.904} C_VEL
LIN {X 0,Y 246.99,Z 374.948,A -85,B 0,C 180,E1 -28479.189,E2 -28479.189} C_VEL
LIN {X 0,Y 251.976,Z 383.805,A -85,B 0,C 180,E1 -28481.248,E2 -28481.248} C_VEL
LIN {X 0,Y 258.337,Z 396.259,A -85,B 0,C 180,E1 -28483.674,E2 -28483.674} C_VEL
LIN {X 0,Y 264.571,Z 410.31,A -85,B 0,C 180,E1 -28485.9,E2 -28485.9} C_VEL
LIN {X 0,Y 267.313,Z 417.455,A -85,B 0,C 180,E1 -28486.856,E2 -28486.856} C_VEL
LIN {X 0,Y 268.587,Z 431.485,A -85,B 0,C 180,E1 -28487.704,E2 -28487.704} C_VEL
LIN {X 0,Y 267.604,Z 447.59,A -85,B 0,C 180,E1 -28488.104,E2 -28488.104} C_VEL
LIN {X 0,Y 266.829,Z 453.447,A -85,B 0,C 180,E1 -28488.14,E2 -28488.14} C_VEL
LIN {X 0,Y 261.638,Z 472.493,A -85,B 0,C 180,E1 -28487.672,E2 -28487.672} C_VEL
LIN {X 0,Y 260.59,Z 478.302,A -85,B 0,C 180,E1 -28487.747,E2 -28487.747} C_VEL
LIN {X 0,Y 258.611,Z 492.38,A -85,B 0,C 180,E1 -28488.303,E2 -28488.303} C_VEL
LIN {X 0,Y 255.977,Z 505.727,A -85,B 0,C 180,E1 -28489.085,E2 -28489.085} C_VEL
LIN {X 0,Y 252.355,Z 518.857,A -85,B 0,C 180,E1 -28490.075,E2 -28490.075} C_VEL
LIN {X 0,Y 248.118,Z 531.541,A -85,B 0,C 180,E1 -28491.353,E2 -28491.353} C_VEL
LIN {X 0,Y 243.164,Z 544.261,A -85,B 0,C 180,E1 -28493.042,E2 -28493.042} C_VEL
LIN {X 0,Y 238.007,Z 555.662,A -85,B 0,C 180,E1 -28494.985,E2 -28494.985} C_VEL
LIN {X 0,Y 232.887,Z 565.882,A -85,B 0,C 180,E1 -28497.228,E2 -28497.228} C_VEL
LIN {X 0,Y 228.088,Z 574.374,A -85,B 0,C 180,E1 -28499.561,E2 -28499.561} C_VEL
LIN {X 0,Y 223.046,Z 582.528,A -85,B 0,C 180,E1 -28502.411,E2 -28502.411} C_VEL
LIN {X 0,Y 218.716,Z 589.142,A -85,B 0,C 180,E1 -28505.402,E2 -28505.402} C_VEL
LIN {X 0,Y 214.721,Z 595.069,A -85,B 0,C 180,E1 -28508.977,E2 -28508.977} C_VEL
LIN {X 0,Y 211.628,Z 599.471,A -85,B 0,C 180,E1 -28512.675,E2 -28512.675} C_VEL
LIN {X 0,Y 209.4,Z 602.468,A -85,B 0,C 180,E1 -28516.463,E2 -28516.463} C_VEL
LIN {X 0,Y 208.138,Z 604.144,A -85,B 0,C 180,E1 -28520.318,E2 -28520.318} C_VEL
LIN {X 0,Y 207.752,Z 604.529,A -85,B 0,C 180,E1 -28524.2,E2 -28524.2} C_VEL
LIN {X 0,Y 208.368,Z 603.631,A -85,B 0,C 180,E1 -28528.078,E2 -28528.078} C_VEL
LIN {X 0,Y 208.936,Z 602.492,A -85,B 0,C 180,E1 -28530.485,E2 -28530.485} C_VEL
LIN {X 0,Y 208.675,Z 606.552,A -85,B 0,C 180,E1 -28532.891,E2 -28532.891} C_VEL
LIN {X 0,Y 208.388,Z 611.677,A -85,B 0,C 180,E1 -28536.761,E2 -28536.761} C_VEL
LIN {X 0,Y 208.638,Z 614.606,A -85,B 0,C 180,E1 -28539.668,E2 -28539.668} C_VEL
LIN {X 0,Y 210.111,Z 617.406,A -85,B 0,C 180,E1 -28543.499,E2 -28543.499} C_VEL
LIN {X 0,Y 212.796,Z 619.015,A -85,B 0,C 180,E1 -28547.337,E2 -28547.337} C_VEL
LIN {X 0,Y 216.29,Z 619.396,A -85,B 0,C 180,E1 -28550.873,E2 -28550.873} C_VEL
LIN {X 0,Y 220.927,Z 618.617,A -85,B 0,C 180,E1 -28554.345,E2 -28554.345} C_VEL
LIN {X 0,Y 226.676,Z 616.644,A -85,B 0,C 180,E1 -28557.618,E2 -28557.618} C_VEL
LIN {X 0,Y 233.076,Z 613.475,A -85,B 0,C 180,E1 -28560.727,E2 -28560.727} C_VEL
LIN {X 0,Y 240.456,Z 609.014,A -85,B 0,C 180,E1 -28563.609,E2 -28563.609} C_VEL
LIN {X 0,Y 248.673,Z 603.137,A -85,B 0,C 180,E1 -28566.269,E2 -28566.269} C_VEL
LIN {X 0,Y 257.54,Z 595.677,A -85,B 0,C 180,E1 -28568.726,E2 -28568.726} C_VEL
LIN {X 0,Y 265.824,Z 587.685,A -85,B 0,C 180,E1 -28570.709,E2 -28570.709} C_VEL
LIN {X 0,Y 274.625,Z 578.037,A -85,B 0,C 180,E1 -28572.528,E2 -28572.528} C_VEL
LIN {X 0,Y 283.444,Z 566.949,A -85,B 0,C 180,E1 -28574.13,E2 -28574.13} C_VEL
LIN {X 0,Y 291.076,Z 555.884,A -85,B 0,C 180,E1 -28575.354,E2 -28575.354} C_VEL
LIN {X 0,Y 298.497,Z 543.372,A -85,B 0,C 180,E1 -28576.431,E2 -28576.431} C_VEL
LIN {X 0,Y 305.833,Z 528.705,A -85,B 0,C 180,E1 -28577.375,E2 -28577.375} C_VEL
LIN {X 0,Y 311.847,Z 513.914,A -85,B 0,C 180,E1 -28578.079,E2 -28578.079} C_VEL
LIN {X 0,Y 316.89,Z 497.98,A -85,B 0,C 180,E1 -28578.666,E2 -28578.666} C_VEL
LIN {X 0,Y 323.484,Z 469.308,A -85,B 0,C 180,E1 -28579.553,E2 -28579.553} C_VEL
LIN {X 0,Y 323.77,Z 467.997,A -85,B 0,C 180,E1 -28579.606,E2 -28579.606} C_VEL
LIN {X 0,Y 323.52,Z 468.209,A -85,B 0,C 180,E1 -28581.541,E2 -28581.541} C_VEL
LIN {X 0,Y 323.533,Z 469.029,A -85,B 0,C 180,E1 -28582.685,E2 -28582.685} C_VEL
LIN {X 0,Y 317.188,Z 496.698,A -85,B 0,C 180,E1 -28583.548,E2 -28583.548} C_VEL
LIN {X 0,Y 313.241,Z 509.462,A -85,B 0,C 180,E1 -28584.029,E2 -28584.029} C_VEL
LIN {X 0,Y 307.85,Z 523.482,A -85,B 0,C 180,E1 -28584.735,E2 -28584.735} C_VEL
LIN {X 0,Y 302.007,Z 535.967,A -85,B 0,C 180,E1 -28585.575,E2 -28585.575} C_VEL
LIN {X 0,Y 295.74,Z 547.38,A -85,B 0,C 180,E1 -28586.531,E2 -28586.531} C_VEL
LIN {X 0,Y 288.485,Z 558.705,A -85,B 0,C 180,E1 -28587.713,E2 -28587.713} C_VEL
LIN {X 0,Y 280.29,Z 569.745,A -85,B 0,C 180,E1 -28589.183,E2 -28589.183} C_VEL
LIN {X 0,Y 271.227,Z 580.263,A -85,B 0,C 180,E1 -28591.039,E2 -28591.039} C_VEL
LIN {X 0,Y 262.565,Z 588.934,A -85,B 0,C 180,E1 -28593.031,E2 -28593.031} C_VEL
LIN {X 0,Y 255.048,Z 595.476,A -85,B 0,C 180,E1 -28595.004,E2 -28595.004} C_VEL
LIN {X 0,Y 246.9,Z 601.659,A -85,B 0,C 180,E1 -28597.481,E2 -28597.481} C_VEL
LIN {X 0,Y 238.892,Z 606.72,A -85,B 0,C 180,E1 -28600.294,E2 -28600.294} C_VEL
LIN {X 0,Y 233.429,Z 609.513,A -85,B 0,C 180,E1 -28602.538,E2 -28602.538} C_VEL
LIN {X 0,Y 226.766,Z 612.122,A -85,B 0,C 180,E1 -28605.694,E2 -28605.694} C_VEL
LIN {X 0,Y 221.072,Z 613.434,A -85,B 0,C 180,E1 -28609.041,E2 -28609.041} C_VEL
LIN {X 0,Y 216.435,Z 613.49,A -85,B 0,C 180,E1 -28612.562,E2 -28612.562} C_VEL
LIN {X 0,Y 212.835,Z 612.315,A -85,B 0,C 180,E1 -28616.226,E2 -28616.226} C_VEL
LIN {X 0,Y 210.15,Z 609.673,A -85,B 0,C 180,E1 -28620.311,E2 -28620.311} C_VEL
LIN {X 0,Y 208.739,Z 606.226,A -85,B 0,C 180,E1 -28623.848,E2 -28623.848} C_VEL
LIN {X 0,Y 207.973,Z 601.123,A -85,B 0,C 180,E1 -28627.742,E2 -28627.742} C_VEL
LIN {X 0,Y 207.909,Z 596.231,A -85,B 0,C 180,E1 -28630.678,E2 -28630.678} C_VEL
LIN {X 0,Y 208.102,Z 589.14,A -85,B 0,C 180,E1 -28634.124,E2 -28634.124} C_VEL
LIN {X 0,Y 208.463,Z 581.621,A -85,B 0,C 180,E1 -28637.098,E2 -28637.098} C_VEL
LIN {X 0,Y 208.951,Z 572.199,A -85,B 0,C 180,E1 -28640.169,E2 -28640.169} C_VEL
LIN {X 0,Y 209.648,Z 561.17,A -85,B 0,C 180,E1 -28643.115,E2 -28643.115} C_VEL
LIN {X 0,Y 210.567,Z 549.731,A -85,B 0,C 180,E1 -28645.623,E2 -28645.623} C_VEL
LIN {X 0,Y 211.75,Z 535.736,A -85,B 0,C 180,E1 -28648.123,E2 -28648.123} C_VEL
LIN {X 0,Y 212.731,Z 523.662,A -85,B 0,C 180,E1 -28649.868,E2 -28649.868} C_VEL
LIN {X 0,Y 213.698,Z 510.938,A -85,B 0,C 180,E1 -28651.355,E2 -28651.355} C_VEL
LIN {X 0,Y 214.743,Z 496.001,A -85,B 0,C 180,E1 -28652.699,E2 -28652.699} C_VEL
LIN {X 0,Y 215.675,Z 480.128,A -85,B 0,C 180,E1 -28653.721,E2 -28653.721} C_VEL
LIN {X 0,Y 219.738,Z 391.23,A -85,B 0,C 180,E1 -28658.44,E2 -28658.44} C_VEL
LIN {X 0,Y 217.424,Z 365.169,A -85,B 0,C 180,E1 -28659.912,E2 -28659.912} C_VEL
LIN {X 0,Y 216.791,Z 358.388,A -85,B 0,C 180,E1 -28660.301,E2 -28660.301} C_VEL
LIN {X 0,Y 214.316,Z 347.728,A -85,B 0,C 180,E1 -28661.011,E2 -28661.011} C_VEL
LIN {X 0,Y 210.935,Z 330.757,A -85,B 0,C 180,E1 -28665.543,E2 -28665.543} C_VEL
LIN {X 0,Y 210.852,Z 330.772,A -85,B 0,C 180,E1 -28670.858,E2 -28670.858} C_VEL
LIN {X 0,Y 210.822,Z 330.758,A -85,B 0,C 180,E1 -28675.605,E2 -28675.605} C_VEL
LIN {X 0,Y 210.875,Z 330.771,A -85,B 0,C 180,E1 -28680.111,E2 -28680.111} C_VEL
LIN {X 0,Y 210.87,Z 330.758,A -85,B 0,C 180,E1 -28682.249,E2 -28682.249} C_VEL
LIN {X 0,Y 211.881,Z 333.653,A -85,B 0,C 180,E1 -28682.576,E2 -28682.576} C_VEL
LIN {X 0,Y 213.401,Z 335.933,A -85,B 0,C 180,E1 -28682.95,E2 -28682.95} C_VEL
LIN {X 0,Y 220.947,Z 349.31,A -85,B 0,C 180,E1 -28684.786,E2 -28684.786} C_VEL
LIN {X 0,Y 227.999,Z 363.504,A -85,B 0,C 180,E1 -28686.427,E2 -28686.427} C_VEL
LIN {X 0,Y 233.011,Z 375.291,A -85,B 0,C 180,E1 -28687.576,E2 -28687.576} C_VEL
LIN {X 0,Y 229.561,Z 455.884,A -85,B 0,C 180,E1 -28689.978,E2 -28689.978} C_VEL
LIN {X 0,Y 228.425,Z 470.332,A -85,B 0,C 180,E1 -28690.749,E2 -28690.749} C_VEL
LIN {X 0,Y 226.941,Z 483.622,A -85,B 0,C 180,E1 -28691.786,E2 -28691.786} C_VEL
LIN {X 0,Y 224.953,Z 497.511,A -85,B 0,C 180,E1 -28693.256,E2 -28693.256} C_VEL
LIN {X 0,Y 222.48,Z 510.03,A -85,B 0,C 180,E1 -28694.941,E2 -28694.941} C_VEL
LIN {X 0,Y 220.002,Z 521.438,A -85,B 0,C 180,E1 -28696.884,E2 -28696.884} C_VEL
LIN {X 0,Y 217.984,Z 530.897,A -85,B 0,C 180,E1 -28698.88,E2 -28698.88} C_VEL
LIN {X 0,Y 215.286,Z 541.49,A -85,B 0,C 180,E1 -28701.577,E2 -28701.577} C_VEL
LIN {X 0,Y 213.198,Z 550.207,A -85,B 0,C 180,E1 -28704.339,E2 -28704.339} C_VEL
LIN {X 0,Y 211.317,Z 557.488,A -85,B 0,C 180,E1 -28707.145,E2 -28707.145} C_VEL
LIN {X 0,Y 210.135,Z 563.918,A -85,B 0,C 180,E1 -28710.21,E2 -28710.21} C_VEL
LIN {X 0,Y 208.931,Z 569.977,A -85,B 0,C 180,E1 -28713.84,E2 -28713.84} C_VEL
LIN {X 0,Y 208.052,Z 574.839,A -85,B 0,C 180,E1 -28717.735,E2 -28717.735} C_VEL
LIN {X 0,Y 207.964,Z 578.191,A -85,B 0,C 180,E1 -28721.654,E2 -28721.654} C_VEL
LIN {X 0,Y 208.274,Z 580.148,A -85,B 0,C 180,E1 -28725.602,E2 -28725.602} C_VEL
LIN {X 0,Y 209.318,Z 580.742,A -85,B 0,C 180,E1 -28729.545,E2 -28729.545} C_VEL
LIN {X 0,Y 211.063,Z 579.975,A -85,B 0,C 180,E1 -28733.463,E2 -28733.463} C_VEL
LIN {X 0,Y 213.63,Z 577.815,A -85,B 0,C 180,E1 -28737.319,E2 -28737.319} C_VEL
LIN {X 0,Y 216.981,Z 574.196,A -85,B 0,C 180,E1 -28741.092,E2 -28741.092} C_VEL
LIN {X 0,Y 221.16,Z 568.993,A -85,B 0,C 180,E1 -28744.75,E2 -28744.75} C_VEL
LIN {X 0,Y 224.828,Z 563.882,A -85,B 0,C 180,E1 -28747.404,E2 -28747.404} C_VEL
LIN {X 0,Y 229.289,Z 557.043,A -85,B 0,C 180,E1 -28750.207,E2 -28750.207} C_VEL
LIN {X 0,Y 234.175,Z 548.737,A -85,B 0,C 180,E1 -28752.874,E2 -28752.874} C_VEL
LIN {X 0,Y 238.98,Z 539.627,A -85,B 0,C 180,E1 -28755.183,E2 -28755.183} C_VEL
LIN {X 0,Y 244.002,Z 528.802,A -85,B 0,C 180,E1 -28757.351,E2 -28757.351} C_VEL
LIN {X 0,Y 248.664,Z 517.107,A -85,B 0,C 180,E1 -28759.195,E2 -28759.195} C_VEL
LIN {X 0,Y 252.654,Z 505.193,A -85,B 0,C 180,E1 -28760.687,E2 -28760.687} C_VEL
LIN {X 0,Y 256.173,Z 492.161,A -85,B 0,C 180,E1 -28761.974,E2 -28761.974} C_VEL
LIN {X 0,Y 258.9,Z 479.283,A -85,B 0,C 180,E1 -28762.942,E2 -28762.942} C_VEL
LIN {X 0,Y 260.997,Z 465.753,A -85,B 0,C 180,E1 -28763.688,E2 -28763.688} C_VEL
LIN {X 0,Y 262.434,Z 451.601,A -85,B 0,C 180,E1 -28764.189,E2 -28764.189} C_VEL
LIN {X 0,Y 265.294,Z 407.682,A -85,B 0,C 180,E1 -28765.278,E2 -28765.278} C_VEL
LIN {X 0,Y 258.923,Z 395.717,A -85,B 0,C 180,E1 -28767.439,E2 -28767.439} C_VEL
LIN {X 0,Y 252.358,Z 384.607,A -85,B 0,C 180,E1 -28769.847,E2 -28769.847} C_VEL
LIN {X 0,Y 245.746,Z 374.538,A -85,B 0,C 180,E1 -28772.512,E2 -28772.512} C_VEL
LIN {X 0,Y 239.785,Z 366.182,A -85,B 0,C 180,E1 -28775.186,E2 -28775.186} C_VEL
LIN {X 0,Y 236.56,Z 361.825,A -85,B 0,C 180,E1 -28776.785,E2 -28776.785} C_VEL
LIN {X 0,Y 233.382,Z 357.638,A -85,B 0,C 180,E1 -28778.483,E2 -28778.483} C_VEL
LIN {X 0,Y 230.541,Z 353.968,A -85,B 0,C 180,E1 -28780.123,E2 -28780.123} C_VEL
LIN {X 0,Y 229.416,Z 352.68,A -85,B 0,C 180,E1 -28780.8,E2 -28780.8} C_VEL
LIN {X 0,Y 226.807,Z 349.573,A -85,B 0,C 180,E1 -28782.476,E2 -28782.476} C_VEL
LIN {X 0,Y 225.937,Z 348.106,A -85,B 0,C 180,E1 -28783.104,E2 -28783.104} C_VEL
LIN {X 0,Y 223.319,Z 345.831,A -85,B 0,C 180,E1 -28784.945,E2 -28784.945} C_VEL
LIN {X 0,Y 221.497,Z 342.57,A -85,B 0,C 180,E1 -28786.513,E2 -28786.513} C_VEL
LIN {X 0,Y 218.7,Z 340.676,A -85,B 0,C 180,E1 -28788.921,E2 -28788.921} C_VEL
LIN {X 0,Y 217.036,Z 337.831,A -85,B 0,C 180,E1 -28790.772,E2 -28790.772} C_VEL
LIN {X 0,Y 216.755,Z 336.882,A -85,B 0,C 180,E1 -28791.17,E2 -28791.17} C_VEL
LIN {X 0,Y 213.283,Z 334.585,A -85,B 0,C 180,E1 -28795.762,E2 -28795.762} C_VEL
LIN {X 0,Y 211.874,Z 331.954,A -85,B 0,C 180,E1 -28798.935,E2 -28798.935} C_VEL
LIN {X 0,Y 211.678,Z 330.663,A -85,B 0,C 180,E1 -28800,E2 -28800} C_VEL
LIN {X 0,Y 211.526,Z 330.681,A -85,B 0,C 180,E1 -28803.797,E2 -28803.797} C_VEL
LIN {X 0,Y 211.334,Z 330.69,A -85,B 0,C 180,E1 -28807.619,E2 -28807.619} C_VEL
LIN {X 0,Y 211.264,Z 331.099,A -85,B 0,C 180,E1 -28809.542,E2 -28809.542} C_VEL
LIN {X 0,Y 211.464,Z 332.054,A -85,B 0,C 180,E1 -28811.342,E2 -28811.342} C_VEL
LIN {X 0,Y 213.277,Z 335.069,A -85,B 0,C 180,E1 -28815.577,E2 -28815.577} C_VEL
LIN {X 0,Y 218.03,Z 340.996,A -85,B 0,C 180,E1 -28821.778,E2 -28821.778} C_VEL
LIN {X 0,Y 222.513,Z 347.316,A -85,B 0,C 180,E1 -28825.898,E2 -28825.898} C_VEL
LIN {X 0,Y 223.837,Z 348.996,A -85,B 0,C 180,E1 -28826.921,E2 -28826.921} C_VEL
LIN {X 0,Y 228.116,Z 355.06,A -85,B 0,C 180,E1 -28829.932,E2 -28829.932} C_VEL
LIN {X 0,Y 233.258,Z 362.719,A -85,B 0,C 180,E1 -28833.048,E2 -28833.048} C_VEL
LIN {X 0,Y 237.411,Z 369.346,A -85,B 0,C 180,E1 -28835.286,E2 -28835.286} C_VEL
LIN {X 0,Y 241.232,Z 375.758,A -85,B 0,C 180,E1 -28837.165,E2 -28837.165} C_VEL
LIN {X 0,Y 245.787,Z 383.593,A -85,B 0,C 180,E1 -28839.22,E2 -28839.22} C_VEL
LIN {X 0,Y 252.268,Z 396.17,A -85,B 0,C 180,E1 -28841.922,E2 -28841.922} C_VEL
LIN {X 0,Y 258.024,Z 408.6,A -85,B 0,C 180,E1 -28844.127,E2 -28844.127} C_VEL
LIN {X 0,Y 262.705,Z 420.37,A -85,B 0,C 180,E1 -28845.847,E2 -28845.847} C_VEL
LIN {X 0,Y 263.758,Z 432.669,A -85,B 0,C 180,E1 -28846.609,E2 -28846.609} C_VEL
LIN {X 0,Y 260.59,Z 478.302,A -85,B 0,C 180,E1 -28847.747,E2 -28847.747} C_VEL
LIN {X 0,Y 259.894,Z 482.164,A -85,B 0,C 180,E1 -28847.824,E2 -28847.824} C_VEL
LIN {X 0,Y 257.452,Z 489.703,A -85,B 0,C 180,E1 -28847.804,E2 -28847.804} C_VEL
LIN {X 0,Y 252.138,Z 502.58,A -85,B 0,C 180,E1 -28847.828,E2 -28847.828} C_VEL
LIN {X 0,Y 250.402,Z 508.069,A -85,B 0,C 180,E1 -28848.101,E2 -28848.101} C_VEL
LIN {X 0,Y 246.389,Z 521.509,A -85,B 0,C 180,E1 -28849.173,E2 -28849.173} C_VEL
LIN {X 0,Y 242.138,Z 533.593,A -85,B 0,C 180,E1 -28850.482,E2 -28850.482} C_VEL
LIN {X 0,Y 237.046,Z 545.83,A -85,B 0,C 180,E1 -28852.189,E2 -28852.189} C_VEL
LIN {X 0,Y 232.238,Z 555.941,A -85,B 0,C 180,E1 -28853.981,E2 -28853.981} C_VEL
LIN {X 0,Y 226.948,Z 566.012,A -85,B 0,C 180,E1 -28856.257,E2 -28856.257} C_VEL
LIN {X 0,Y 222,Z 574.412,A -85,B 0,C 180,E1 -28858.633,E2 -28858.633} C_VEL
LIN {X 0,Y 216.753,Z 582.475,A -85,B 0,C 180,E1 -28861.539,E2 -28861.539} C_VEL
LIN {X 0,Y 212.253,Z 589.016,A -85,B 0,C 180,E1 -28864.601,E2 -28864.601} C_VEL
LIN {X 0,Y 208.089,Z 594.876,A -85,B 0,C 180,E1 -28868.273,E2 -28868.273} C_VEL
LIN {X 0,Y 204.836,Z 599.216,A -85,B 0,C 180,E1 -28872.081,E2 -28872.081} C_VEL
LIN {X 0,Y 202.469,Z 602.152,A -85,B 0,C 180,E1 -28875.991,E2 -28875.991} C_VEL
LIN {X 0,Y 201.116,Z 603.771,A -85,B 0,C 180,E1 -28879.977,E2 -28879.977} C_VEL
LIN {X 0,Y 200.659,Z 604.097,A -85,B 0,C 180,E1 -28883.994,E2 -28883.994} C_VEL
LIN {X 0,Y 201.256,Z 603.143,A -85,B 0,C 180,E1 -28888.01,E2 -28888.01} C_VEL
LIN {X 0,Y 202.014,Z 601.676,A -85,B 0,C 180,E1 -28890.998,E2 -28890.998} C_VEL
LIN {X 0,Y 201.615,Z 606.499,A -85,B 0,C 180,E1 -28893.989,E2 -28893.989} C_VEL
LIN {X 0,Y 201.516,Z 611.542,A -85,B 0,C 180,E1 -28897.997,E2 -28897.997} C_VEL
LIN {X 0,Y 202.39,Z 615.225,A -85,B 0,C 180,E1 -28901.99,E2 -28901.99} C_VEL
LIN {X 0,Y 204.539,Z 617.692,A -85,B 0,C 180,E1 -28905.905,E2 -28905.905} C_VEL
LIN {X 0,Y 207.703,Z 618.961,A -85,B 0,C 180,E1 -28909.713,E2 -28909.713} C_VEL
LIN {X 0,Y 211.926,Z 619.078,A -85,B 0,C 180,E1 -28913.371,E2 -28913.371} C_VEL
LIN {X 0,Y 217.305,Z 618.037,A -85,B 0,C 180,E1 -28916.829,E2 -28916.829} C_VEL
LIN {X 0,Y 223.722,Z 615.806,A -85,B 0,C 180,E1 -28920.067,E2 -28920.067} C_VEL
LIN {X 0,Y 227.048,Z 614.265,A -85,B 0,C 180,E1 -28921.636,E2 -28921.636} C_VEL
LIN {X 0,Y 234.661,Z 610.188,A -85,B 0,C 180,E1 -28924.555,E2 -28924.555} C_VEL
LIN {X 0,Y 243.097,Z 604.736,A -85,B 0,C 180,E1 -28927.239,E2 -28927.239} C_VEL
LIN {X 0,Y 252.217,Z 597.789,A -85,B 0,C 180,E1 -28929.702,E2 -28929.702} C_VEL
LIN {X 0,Y 260.695,Z 590.345,A -85,B 0,C 180,E1 -28931.686,E2 -28931.686} C_VEL
LIN {X 0,Y 269.703,Z 581.332,A -85,B 0,C 180,E1 -28933.494,E2 -28933.494} C_VEL
LIN {X 0,Y 278.999,Z 570.591,A -85,B 0,C 180,E1 -28935.147,E2 -28935.147} C_VEL
LIN {X 0,Y 287.456,Z 559.237,A -85,B 0,C 180,E1 -28936.466,E2 -28936.466} C_VEL
LIN {X 0,Y 295.438,Z 546.859,A -85,B 0,C 180,E1 -28937.56,E2 -28937.56} C_VEL
LIN {X 0,Y 302.9,Z 533.166,A -85,B 0,C 180,E1 -28938.478,E2 -28938.478} C_VEL
LIN {X 0,Y 309.041,Z 519.546,A -85,B 0,C 180,E1 -28939.156,E2 -28939.156} C_VEL
LIN {X 0,Y 314.6,Z 504.111,A -85,B 0,C 180,E1 -28939.766,E2 -28939.766} C_VEL
LIN {X 0,Y 319.142,Z 487.364,A -85,B 0,C 180,E1 -28940.299,E2 -28940.299} C_VEL
LIN {X 0,Y 321.973,Z 474.936,A -85,B 0,C 180,E1 -28940.672,E2 -28940.672} C_VEL
LIN {X 0,Y 321.915,Z 475.165,A -85,B 0,C 180,E1 -28941.568,E2 -28941.568} C_VEL
LIN {X 0,Y 316.442,Z 497.856,A -85,B 0,C 180,E1 -28942.288,E2 -28942.288} C_VEL
LIN {X 0,Y 311.756,Z 512.204,A -85,B 0,C 180,E1 -28942.822,E2 -28942.822} C_VEL
LIN {X 0,Y 306.225,Z 525.741,A -85,B 0,C 180,E1 -28943.508,E2 -28943.508} C_VEL
LIN {X 0,Y 300.236,Z 537.837,A -85,B 0,C 180,E1 -28944.321,E2 -28944.321} C_VEL
LIN {X 0,Y 293.574,Z 549.309,A -85,B 0,C 180,E1 -28945.273,E2 -28945.273} C_VEL
LIN {X 0,Y 285.603,Z 560.997,A -85,B 0,C 180,E1 -28946.502,E2 -28946.502} C_VEL
LIN {X 0,Y 277.12,Z 571.703,A -85,B 0,C 180,E1 -28947.941,E2 -28947.941} C_VEL
LIN {X 0,Y 268.992,Z 580.67,A -85,B 0,C 180,E1 -28949.519,E2 -28949.519} C_VEL
LIN {X 0,Y 260.067,Z 589.208,A -85,B 0,C 180,E1 -28951.441,E2 -28951.441} C_VEL
LIN {X 0,Y 251.558,Z 596.236,A -85,B 0,C 180,E1 -28953.544,E2 -28953.544} C_VEL
LIN {X 0,Y 242.518,Z 602.607,A -85,B 0,C 180,E1 -28956.15,E2 -28956.15} C_VEL
LIN {X 0,Y 234.133,Z 607.44,A -85,B 0,C 180,E1 -28958.961,E2 -28958.961} C_VEL
LIN {X 0,Y 226.608,Z 610.85,A -85,B 0,C 180,E1 -28961.995,E2 -28961.995} C_VEL
LIN {X 0,Y 219.807,Z 612.966,A -85,B 0,C 180,E1 -28965.23,E2 -28965.23} C_VEL
LIN {X 0,Y 214.011,Z 613.81,A -85,B 0,C 180,E1 -28968.675,E2 -28968.675} C_VEL
LIN {X 0,Y 209.309,Z 613.422,A -85,B 0,C 180,E1 -28972.307,E2 -28972.307} C_VEL
LIN {X 0,Y 205.702,Z 611.82,A -85,B 0,C 180,E1 -28976.095,E2 -28976.095} C_VEL
LIN {X 0,Y 203.143,Z 608.905,A -85,B 0,C 180,E1 -28980.1,E2 -28980.1} C_VEL
LIN {X 0,Y 201.656,Z 604.876,A -85,B 0,C 180,E1 -28983.983,E2 -28983.983} C_VEL
LIN {X 0,Y 200.989,Z 599.304,A -85,B 0,C 180,E1 -28988.013,E2 -28988.013} C_VEL
LIN {X 0,Y 200.956,Z 593.04,A -85,B 0,C 180,E1 -28991.561,E2 -28991.561} C_VEL
LIN {X 0,Y 201.272,Z 585.195,A -85,B 0,C 180,E1 -28995.13,E2 -28995.13} C_VEL
LIN {X 0,Y 201.673,Z 576.836,A -85,B 0,C 180,E1 -28998.215,E2 -28998.215} C_VEL
LIN {X 0,Y 202.21,Z 566.981,A -85,B 0,C 180,E1 -29001.222,E2 -29001.222} C_VEL
LIN {X 0,Y 202.954,Z 556.33,A -85,B 0,C 180,E1 -29003.924,E2 -29003.924} C_VEL
LIN {X 0,Y 203.795,Z 545.201,A -85,B 0,C 180,E1 -29006.264,E2 -29006.264} C_VEL
LIN {X 0,Y 204.828,Z 533.572,A -85,B 0,C 180,E1 -29008.298,E2 -29008.298} C_VEL
LIN {X 0,Y 205.962,Z 519.824,A -85,B 0,C 180,E1 -29010.248,E2 -29010.248} C_VEL
LIN {X 0,Y 207.103,Z 504.268,A -85,B 0,C 180,E1 -29011.972,E2 -29011.972} C_VEL
LIN {X 0,Y 208.114,Z 488.668,A -85,B 0,C 180,E1 -29013.228,E2 -29013.228} C_VEL
LIN {X 0,Y 209.868,Z 449.978,A -85,B 0,C 180,E1 -29015.443,E2 -29015.443} C_VEL
LIN {X 0,Y 212.681,Z 391.706,A -85,B 0,C 180,E1 -29018.634,E2 -29018.634} C_VEL
LIN {X 0,Y 210.275,Z 363.967,A -85,B 0,C 180,E1 -29020.262,E2 -29020.262} C_VEL
LIN {X 0,Y 209.746,Z 359.157,A -85,B 0,C 180,E1 -29020.553,E2 -29020.553} C_VEL
LIN {X 0,Y 207.059,Z 347.737,A -85,B 0,C 180,E1 -29021.355,E2 -29021.355} C_VEL
LIN {X 0,Y 203.904,Z 331.633,A -85,B 0,C 180,E1 -29025.818,E2 -29025.818} C_VEL
LIN {X 0,Y 203.777,Z 331.655,A -85,B 0,C 180,E1 -29029.22,E2 -29029.22} C_VEL
LIN {X 0,Y 203.782,Z 331.66,A -85,B 0,C 180,E1 -29032.238,E2 -29032.238} C_VEL
LIN {X 0,Y 203.771,Z 331.636,A -85,B 0,C 180,E1 -29036.629,E2 -29036.629} C_VEL
LIN {X 0,Y 203.861,Z 331.789,A -85,B 0,C 180,E1 -29040.923,E2 -29040.923} C_VEL
LIN {X 0,Y 204.987,Z 334.735,A -85,B 0,C 180,E1 -29041.28,E2 -29041.28} C_VEL
LIN {X 0,Y 206.429,Z 336.945,A -85,B 0,C 180,E1 -29041.663,E2 -29041.663} C_VEL
LIN {X 0,Y 213.676,Z 349.381,A -85,B 0,C 180,E1 -29043.539,E2 -29043.539} C_VEL
LIN {X 0,Y 221.897,Z 365.615,A -85,B 0,C 180,E1 -29045.557,E2 -29045.557} C_VEL
LIN {X 0,Y 226.797,Z 377.1,A -85,B 0,C 180,E1 -29046.74,E2 -29046.74} C_VEL
LIN {X 0,Y 223.292,Z 456.193,A -85,B 0,C 180,E1 -29049.151,E2 -29049.151} C_VEL
LIN {X 0,Y 222.182,Z 469.927,A -85,B 0,C 180,E1 -29049.885,E2 -29049.885} C_VEL
LIN {X 0,Y 220.574,Z 483.981,A -85,B 0,C 180,E1 -29051,E2 -29051} C_VEL
LIN {X 0,Y 218.508,Z 497.88,A -85,B 0,C 180,E1 -29052.507,E2 -29052.507} C_VEL
LIN {X 0,Y 215.927,Z 510.414,A -85,B 0,C 180,E1 -29054.231,E2 -29054.231} C_VEL
LIN {X 0,Y 213.378,Z 521.822,A -85,B 0,C 180,E1 -29056.227,E2 -29056.227} C_VEL
LIN {X 0,Y 211.021,Z 532.262,A -85,B 0,C 180,E1 -29058.508,E2 -29058.508} C_VEL
LIN {X 0,Y 208.261,Z 542.698,A -85,B 0,C 180,E1 -29061.29,E2 -29061.29} C_VEL
LIN {X 0,Y 206.143,Z 551.279,A -85,B 0,C 180,E1 -29064.145,E2 -29064.145} C_VEL
LIN {X 0,Y 204.243,Z 558.443,A -85,B 0,C 180,E1 -29067.047,E2 -29067.047} C_VEL
LIN {X 0,Y 203.091,Z 564.368,A -85,B 0,C 180,E1 -29069.995,E2 -29069.995} C_VEL
LIN {X 0,Y 202.071,Z 569.304,A -85,B 0,C 180,E1 -29072.976,E2 -29072.976} C_VEL
LIN {X 0,Y 201.075,Z 574.434,A -85,B 0,C 180,E1 -29076.998,E2 -29076.998} C_VEL
LIN {X 0,Y 200.842,Z 577.308,A -85,B 0,C 180,E1 -29080.037,E2 -29080.037} C_VEL
LIN {X 0,Y 201.014,Z 579.86,A -85,B 0,C 180,E1 -29084.113,E2 -29084.113} C_VEL
LIN {X 0,Y 201.768,Z 581.058,A -85,B 0,C 180,E1 -29088.201,E2 -29088.201} C_VEL
LIN {X 0,Y 203.331,Z 580.893,A -85,B 0,C 180,E1 -29092.262,E2 -29092.262} C_VEL
LIN {X 0,Y 205.64,Z 579.357,A -85,B 0,C 180,E1 -29096.277,E2 -29096.277} C_VEL
LIN {X 0,Y 208.835,Z 576.396,A -85,B 0,C 180,E1 -29100.2,E2 -29100.2} C_VEL
LIN {X 0,Y 212.841,Z 571.912,A -85,B 0,C 180,E1 -29104.012,E2 -29104.012} C_VEL
LIN {X 0,Y 216.428,Z 567.402,A -85,B 0,C 180,E1 -29106.773,E2 -29106.773} C_VEL
LIN {X 0,Y 221.119,Z 560.861,A -85,B 0,C 180,E1 -29109.883,E2 -29109.883} C_VEL
LIN {X 0,Y 226.416,Z 552.615,A -85,B 0,C 180,E1 -29112.883,E2 -29112.883} C_VEL
LIN {X 0,Y 231.406,Z 543.92,A -85,B 0,C 180,E1 -29115.336,E2 -29115.336} C_VEL
LIN {X 0,Y 235.912,Z 535.151,A -85,B 0,C 180,E1 -29117.322,E2 -29117.322} C_VEL
LIN {X 0,Y 240.561,Z 524.9,A -85,B 0,C 180,E1 -29119.197,E2 -29119.197} C_VEL
LIN {X 0,Y 245.048,Z 513.272,A -85,B 0,C 180,E1 -29120.904,E2 -29120.904} C_VEL
LIN {X 0,Y 248.943,Z 501.192,A -85,B 0,C 180,E1 -29122.304,E2 -29122.304} C_VEL
LIN {X 0,Y 252.198,Z 488.404,A -85,B 0,C 180,E1 -29123.477,E2 -29123.477} C_VEL
LIN {X 0,Y 254.939,Z 474.81,A -85,B 0,C 180,E1 -29124.391,E2 -29124.391} C_VEL
LIN {X 0,Y 256.806,Z 461.35,A -85,B 0,C 180,E1 -29125.044,E2 -29125.044} C_VEL
LIN {X 0,Y 258.272,Z 442.862,A -85,B 0,C 180,E1 -29125.593,E2 -29125.593} C_VEL
LIN {X 0,Y 260.454,Z 410.461,A -85,B 0,C 180,E1 -29126.395,E2 -29126.395} C_VEL
LIN {X 0,Y 254.218,Z 398.734,A -85,B 0,C 180,E1 -29128.631,E2 -29128.631} C_VEL
LIN {X 0,Y 247.675,Z 387.645,A -85,B 0,C 180,E1 -29131.19,E2 -29131.19} C_VEL
LIN {X 0,Y 240.737,Z 377.036,A -85,B 0,C 180,E1 -29134.201,E2 -29134.201} C_VEL
LIN {X 0,Y 234.621,Z 368.485,A -85,B 0,C 180,E1 -29137.221,E2 -29137.221} C_VEL
LIN {X 0,Y 231.141,Z 363.882,A -85,B 0,C 180,E1 -29139.141,E2 -29139.141} C_VEL
LIN {X 0,Y 227.658,Z 359.302,A -85,B 0,C 180,E1 -29141.261,E2 -29141.261} C_VEL
LIN {X 0,Y 224.882,Z 355.939,A -85,B 0,C 180,E1 -29143.109,E2 -29143.109} C_VEL
LIN {X 0,Y 224.137,Z 354.709,A -85,B 0,C 180,E1 -29143.665,E2 -29143.665} C_VEL
LIN {X 0,Y 221.472,Z 352.138,A -85,B 0,C 180,E1 -29145.637,E2 -29145.637} C_VEL
LIN {X 0,Y 219.813,Z 349.309,A -85,B 0,C 180,E1 -29147.111,E2 -29147.111} C_VEL
LIN {X 0,Y 217.194,Z 347.273,A -85,B 0,C 180,E1 -29149.49,E2 -29149.49} C_VEL
LIN {X 0,Y 215.522,Z 344.257,A -85,B 0,C 180,E1 -29151.473,E2 -29151.473} C_VEL
LIN {X 0,Y 215.078,Z 343.538,A -85,B 0,C 180,E1 -29152.044,E2 -29152.044} C_VEL
LIN {X 0,Y 212.143,Z 341.396,A -85,B 0,C 180,E1 -29156.214,E2 -29156.214} C_VEL
LIN {X 0,Y 210.827,Z 338.749,A -85,B 0,C 180,E1 -29159.405,E2 -29159.405} C_VEL
LIN {X 0,Y 210.64,Z 337.705,A -85,B 0,C 180,E1 -29160.238,E2 -29160.238} C_VEL
LIN {X 0,Y 209.974,Z 337.793,A -85,B 0,C 180,E1 -29168.634,E2 -29168.634} C_VEL
LIN {X 0,Y 210.454,Z 338.917,A -85,B 0,C 180,E1 -29170.912,E2 -29170.912} C_VEL
LIN {X 0,Y 212.692,Z 342.758,A -85,B 0,C 180,E1 -29176.133,E2 -29176.133} C_VEL
LIN {X 0,Y 216.606,Z 347.692,A -85,B 0,C 180,E1 -29181.271,E2 -29181.271} C_VEL
LIN {X 0,Y 221.031,Z 354.074,A -85,B 0,C 180,E1 -29185.486,E2 -29185.486} C_VEL
LIN {X 0,Y 222.004,Z 355.435,A -85,B 0,C 180,E1 -29186.276,E2 -29186.276} C_VEL
LIN {X 0,Y 226.87,Z 362.621,A -85,B 0,C 180,E1 -29189.81,E2 -29189.81} C_VEL
LIN {X 0,Y 230.909,Z 368.796,A -85,B 0,C 180,E1 -29192.333,E2 -29192.333} C_VEL
LIN {X 0,Y 234.893,Z 375.327,A -85,B 0,C 180,E1 -29194.577,E2 -29194.577} C_VEL
LIN {X 0,Y 240.028,Z 384.066,A -85,B 0,C 180,E1 -29197.169,E2 -29197.169} C_VEL
LIN {X 0,Y 245.822,Z 395.168,A -85,B 0,C 180,E1 -29199.822,E2 -29199.822} C_VEL
LIN {X 0,Y 251.417,Z 406.812,A -85,B 0,C 180,E1 -29202.164,E2 -29202.164} C_VEL
LIN {X 0,Y 256.455,Z 418.808,A -85,B 0,C 180,E1 -29204.145,E2 -29204.145} C_VEL
LIN {X 0,Y 258.257,Z 423.778,A -85,B 0,C 180,E1 -29204.844,E2 -29204.844} C_VEL
LIN {X 0,Y 258.985,Z 434.168,A -85,B 0,C 180,E1 -29205.475,E2 -29205.475} C_VEL
LIN {X 0,Y 255.768,Z 478.592,A -85,B 0,C 180,E1 -29206.6,E2 -29206.6} C_VEL
LIN {X 0,Y 253.686,Z 492.698,A -85,B 0,C 180,E1 -29207.169,E2 -29207.169} C_VEL
LIN {X 0,Y 250.968,Z 505.858,A -85,B 0,C 180,E1 -29207.952,E2 -29207.952} C_VEL
LIN {X 0,Y 250.402,Z 508.069,A -85,B 0,C 180,E1 -29208.101,E2 -29208.101} C_VEL
LIN {X 0,Y 248.49,Z 513.516,A -85,B 0,C 180,E1 -29208.393,E2 -29208.393} C_VEL
LIN {X 0,Y 243.741,Z 522.164,A -85,B 0,C 180,E1 -29208.656,E2 -29208.656} C_VEL
LIN {X 0,Y 238.655,Z 530.491,A -85,B 0,C 180,E1 -29209.053,E2 -29209.053} C_VEL
LIN {X 0,Y 236.231,Z 535.427,A -85,B 0,C 180,E1 -29209.561,E2 -29209.561} C_VEL
LIN {X 0,Y 230.988,Z 547.27,A -85,B 0,C 180,E1 -29211.292,E2 -29211.292} C_VEL
LIN {X 0,Y 225.624,Z 557.961,A -85,B 0,C 180,E1 -29213.307,E2 -29213.307} C_VEL
LIN {X 0,Y 220.127,Z 567.777,A -85,B 0,C 180,E1 -29215.672,E2 -29215.672} C_VEL
LIN {X 0,Y 214.342,Z 576.918,A -85,B 0,C 180,E1 -29218.482,E2 -29218.482} C_VEL
LIN {X 0,Y 209.833,Z 583.444,A -85,B 0,C 180,E1 -29221.057,E2 -29221.057} C_VEL
LIN {X 0,Y 204.648,Z 590.523,A -85,B 0,C 180,E1 -29224.675,E2 -29224.675} C_VEL
LIN {X 0,Y 200.545,Z 595.915,A -85,B 0,C 180,E1 -29228.491,E2 -29228.491} C_VEL
LIN {X 0,Y 198.066,Z 598.96,A -85,B 0,C 180,E1 -29231.447,E2 -29231.447} C_VEL
LIN {X 0,Y 195.544,Z 601.837,A -85,B 0,C 180,E1 -29235.484,E2 -29235.484} C_VEL
LIN {X 0,Y 194.09,Z 603.397,A -85,B 0,C 180,E1 -29239.61,E2 -29239.61} C_VEL
LIN {X 0,Y 193.571,Z 603.667,A -85,B 0,C 180,E1 -29243.773,E2 -29243.773} C_VEL
LIN {X 0,Y 194.151,Z 602.655,A -85,B 0,C 180,E1 -29247.938,E2 -29247.938} C_VEL
LIN {X 0,Y 195.063,Z 600.771,A -85,B 0,C 180,E1 -29251.548,E2 -29251.548} C_VEL
LIN {X 0,Y 194.703,Z 604.949,A -85,B 0,C 180,E1 -29254.131,E2 -29254.131} C_VEL
LIN {X 0,Y 194.582,Z 610.276,A -85,B 0,C 180,E1 -29258.284,E2 -29258.284} C_VEL
LIN {X 0,Y 195.501,Z 614.235,A -85,B 0,C 180,E1 -29262.419,E2 -29262.419} C_VEL
LIN {X 0,Y 197.741,Z 616.986,A -85,B 0,C 180,E1 -29266.467,E2 -29266.467} C_VEL
LIN {X 0,Y 201.047,Z 618.556,A -85,B 0,C 180,E1 -29270.394,E2 -29270.394} C_VEL
LIN {X 0,Y 205.432,Z 618.971,A -85,B 0,C 180,E1 -29274.156,E2 -29274.156} C_VEL
LIN {X 0,Y 211.009,Z 618.24,A -85,B 0,C 180,E1 -29277.697,E2 -29277.697} C_VEL
LIN {X 0,Y 217.642,Z 616.351,A -85,B 0,C 180,E1 -29280.998,E2 -29280.998} C_VEL
LIN {X 0,Y 221.066,Z 614.983,A -85,B 0,C 180,E1 -29282.596,E2 -29282.596} C_VEL
LIN {X 0,Y 228.916,Z 611.293,A -85,B 0,C 180,E1 -29285.551,E2 -29285.551} C_VEL
LIN {X 0,Y 237.589,Z 606.294,A -85,B 0,C 180,E1 -29288.255,E2 -29288.255} C_VEL
LIN {X 0,Y 246.952,Z 599.869,A -85,B 0,C 180,E1 -29290.724,E2 -29290.724} C_VEL
LIN {X 0,Y 255.62,Z 592.922,A -85,B 0,C 180,E1 -29292.707,E2 -29292.707} C_VEL
LIN {X 0,Y 265.087,Z 584.239,A -85,B 0,C 180,E1 -29294.555,E2 -29294.555} C_VEL
LIN {X 0,Y 274.306,Z 574.444,A -85,B 0,C 180,E1 -29296.141,E2 -29296.141} C_VEL
LIN {X 0,Y 282.892,Z 563.987,A -85,B 0,C 180,E1 -29297.448,E2 -29297.448} C_VEL
LIN {X 0,Y 291.733,Z 551.487,A -85,B 0,C 180,E1 -29298.621,E2 -29298.621} C_VEL
LIN {X 0,Y 299.319,Z 538.895,A -85,B 0,C 180,E1 -29299.516,E2 -29299.516} C_VEL
LIN {X 0,Y 305.85,Z 525.971,A -85,B 0,C 180,E1 -29300.21,E2 -29300.21} C_VEL
LIN {X 0,Y 311.528,Z 512.344,A -85,B 0,C 180,E1 -29300.781,E2 -29300.781} C_VEL
LIN {X 0,Y 314.936,Z 502.513,A -85,B 0,C 180,E1 -29301.121,E2 -29301.121} C_VEL
LIN {X 0,Y 309.553,Z 517.308,A -85,B 0,C 180,E1 -29301.725,E2 -29301.725} C_VEL
LIN {X 0,Y 303.308,Z 531.036,A -85,B 0,C 180,E1 -29302.448,E2 -29302.448} C_VEL
LIN {X 0,Y 295.508,Z 545.102,A -85,B 0,C 180,E1 -29303.453,E2 -29303.453} C_VEL
LIN {X 0,Y 287.238,Z 557.514,A -85,B 0,C 180,E1 -29304.609,E2 -29304.609} C_VEL
LIN {X 0,Y 278.285,Z 569.01,A -85,B 0,C 180,E1 -29305.986,E2 -29305.986} C_VEL
LIN {X 0,Y 269.952,Z 578.219,A -85,B 0,C 180,E1 -29307.425,E2 -29307.425} C_VEL
LIN {X 0,Y 260.433,Z 587.283,A -85,B 0,C 180,E1 -29309.269,E2 -29309.269} C_VEL
LIN {X 0,Y 252.656,Z 593.75,A -85,B 0,C 180,E1 -29310.977,E2 -29310.977} C_VEL
LIN {X 0,Y 245.243,Z 599.128,A -85,B 0,C 180,E1 -29312.807,E2 -29312.807} C_VEL
LIN {X 0,Y 236.034,Z 604.868,A -85,B 0,C 180,E1 -29315.452,E2 -29315.452} C_VEL
LIN {X 0,Y 227.477,Z 609.142,A -85,B 0,C 180,E1 -29318.315,E2 -29318.315} C_VEL
LIN {X 0,Y 219.77,Z 612.033,A -85,B 0,C 180,E1 -29321.415,E2 -29321.415} C_VEL
LIN {X 0,Y 212.854,Z 613.661,A -85,B 0,C 180,E1 -29324.736,E2 -29324.736} C_VEL
LIN {X 0,Y 206.956,Z 614.043,A -85,B 0,C 180,E1 -29328.283,E2 -29328.283} C_VEL
LIN {X 0,Y 202.205,Z 613.208,A -85,B 0,C 180,E1 -29332.035,E2 -29332.035} C_VEL
LIN {X 0,Y 198.578,Z 611.177,A -85,B 0,C 180,E1 -29335.955,E2 -29335.955} C_VEL
LIN {X 0,Y 196.091,Z 607.932,A -85,B 0,C 180,E1 -29340,E2 -29340} C_VEL
LIN {X 0,Y 194.586,Z 603.362,A -85,B 0,C 180,E1 -29344.128,E2 -29344.128} C_VEL
LIN {X 0,Y 194.002,Z 597.304,A -85,B 0,C 180,E1 -29348.304,E2 -29348.304} C_VEL
LIN {X 0,Y 194.051,Z 590.577,A -85,B 0,C 180,E1 -29351.979,E2 -29351.979} C_VEL
LIN {X 0,Y 194.354,Z 583.481,A -85,B 0,C 180,E1 -29355.146,E2 -29355.146} C_VEL
LIN {X 0,Y 194.73,Z 574.766,A -85,B 0,C 180,E1 -29358.345,E2 -29358.345} C_VEL
LIN {X 0,Y 195.316,Z 564.301,A -85,B 0,C 180,E1 -29361.511,E2 -29361.511} C_VEL
LIN {X 0,Y 196.18,Z 552.129,A -85,B 0,C 180,E1 -29364.523,E2 -29364.523} C_VEL
LIN {X 0,Y 197.224,Z 539.23,A -85,B 0,C 180,E1 -29367.12,E2 -29367.12} C_VEL
LIN {X 0,Y 198.433,Z 524.744,A -85,B 0,C 180,E1 -29369.456,E2 -29369.456} C_VEL
LIN {X 0,Y 199.492,Z 511.151,A -85,B 0,C 180,E1 -29371.191,E2 -29371.191} C_VEL
LIN {X 0,Y 200.56,Z 495.881,A -85,B 0,C 180,E1 -29372.667,E2 -29372.667} C_VEL
LIN {X 0,Y 201.51,Z 479.593,A -85,B 0,C 180,E1 -29373.79,E2 -29373.79} C_VEL
LIN {X 0,Y 205.645,Z 392.553,A -85,B 0,C 180,E1 -29378.812,E2 -29378.812} C_VEL
LIN {X 0,Y 203.237,Z 363.894,A -85,B 0,C 180,E1 -29380.544,E2 -29380.544} C_VEL
LIN {X 0,Y 202.252,Z 358.101,A -85,B 0,C 180,E1 -29380.92,E2 -29380.92} C_VEL
LIN {X 0,Y 199.921,Z 347.927,A -85,B 0,C 180,E1 -29381.654,E2 -29381.654} C_VEL
LIN {X 0,Y 196.836,Z 332.514,A -85,B 0,C 180,E1 -29386.073,E2 -29386.073} C_VEL
LIN {X 0,Y 196.746,Z 332.533,A -85,B 0,C 180,E1 -29391.558,E2 -29391.558} C_VEL
LIN {X 0,Y 196.723,Z 332.513,A -85,B 0,C 180,E1 -29395.266,E2 -29395.266} C_VEL
LIN {X 0,Y 196.772,Z 332.533,A -85,B 0,C 180,E1 -29399.383,E2 -29399.383} C_VEL
LIN {X 0,Y 197.879,Z 335.509,A -85,B 0,C 180,E1 -29399.811,E2 -29399.811} C_VEL
LIN {X 0,Y 199.44,Z 337.667,A -85,B 0,C 180,E1 -29400.249,E2 -29400.249} C_VEL
LIN {X 0,Y 208.532,Z 353.296,A -85,B 0,C 180,E1 -29402.753,E2 -29402.753} C_VEL
LIN {X 0,Y 216.572,Z 369.377,A -85,B 0,C 180,E1 -29404.828,E2 -29404.828} C_VEL
LIN {X 0,Y 220.623,Z 378.969,A -85,B 0,C 180,E1 -29405.857,E2 -29405.857} C_VEL
LIN {X 0,Y 217.065,Z 456.505,A -85,B 0,C 180,E1 -29408.275,E2 -29408.275} C_VEL
LIN {X 0,Y 215.92,Z 470.27,A -85,B 0,C 180,E1 -29409.027,E2 -29409.027} C_VEL
LIN {X 0,Y 214.25,Z 484.34,A -85,B 0,C 180,E1 -29410.168,E2 -29410.168} C_VEL
LIN {X 0,Y 212.079,Z 498.258,A -85,B 0,C 180,E1 -29411.709,E2 -29411.709} C_VEL
LIN {X 0,Y 209.41,Z 510.798,A -85,B 0,C 180,E1 -29413.478,E2 -29413.478} C_VEL
LIN {X 0,Y 206.788,Z 522.206,A -85,B 0,C 180,E1 -29415.529,E2 -29415.529} C_VEL
LIN {X 0,Y 204.576,Z 531.679,A -85,B 0,C 180,E1 -29417.639,E2 -29417.639} C_VEL
LIN {X 0,Y 201.677,Z 542.279,A -85,B 0,C 180,E1 -29420.5,E2 -29420.5} C_VEL
LIN {X 0,Y 199.411,Z 551.002,A -85,B 0,C 180,E1 -29423.44,E2 -29423.44} C_VEL
LIN {X 0,Y 197.396,Z 558.287,A -85,B 0,C 180,E1 -29426.435,E2 -29426.435} C_VEL
LIN {X 0,Y 195.975,Z 565.224,A -85,B 0,C 180,E1 -29429.995,E2 -29429.995} C_VEL
LIN {X 0,Y 194.949,Z 570.068,A -85,B 0,C 180,E1 -29433.084,E2 -29433.084} C_VEL
LIN {X 0,Y 193.946,Z 575.114,A -85,B 0,C 180,E1 -29437.257,E2 -29437.257} C_VEL
LIN {X 0,Y 193.739,Z 577.907,A -85,B 0,C 180,E1 -29440.409,E2 -29440.409} C_VEL
LIN {X 0,Y 193.98,Z 580.382,A -85,B 0,C 180,E1 -29444.636,E2 -29444.636} C_VEL
LIN {X 0,Y 194.855,Z 581.502,A -85,B 0,C 180,E1 -29448.871,E2 -29448.871} C_VEL
LIN {X 0,Y 196.583,Z 581.258,A -85,B 0,C 180,E1 -29453.069,E2 -29453.069} C_VEL
LIN {X 0,Y 199.096,Z 579.643,A -85,B 0,C 180,E1 -29457.211,E2 -29457.211} C_VEL
LIN {X 0,Y 202.515,Z 576.601,A -85,B 0,C 180,E1 -29461.246,E2 -29461.246} C_VEL
LIN {X 0,Y 205.642,Z 573.278,A -85,B 0,C 180,E1 -29464.189,E2 -29464.189} C_VEL
LIN {X 0,Y 210.595,Z 567.43,A -85,B 0,C 180,E1 -29467.968,E2 -29467.968} C_VEL
LIN {X 0,Y 214.807,Z 561.788,A -85,B 0,C 180,E1 -29470.698,E2 -29470.698} C_VEL
LIN {X 0,Y 220.288,Z 553.695,A -85,B 0,C 180,E1 -29473.748,E2 -29473.748} C_VEL
LIN {X 0,Y 225.419,Z 545.154,A -85,B 0,C 180,E1 -29476.25,E2 -29476.25} C_VEL
LIN {X 0,Y 230.961,Z 534.753,A -85,B 0,C 180,E1 -29478.635,E2 -29478.635} C_VEL
LIN {X 0,Y 235.854,Z 524.195,A -85,B 0,C 180,E1 -29480.54,E2 -29480.54} C_VEL
LIN {X 0,Y 240.335,Z 512.701,A -85,B 0,C 180,E1 -29482.211,E2 -29482.211} C_VEL
LIN {X 0,Y 244.496,Z 499.86,A -85,B 0,C 180,E1 -29483.674,E2 -29483.674} C_VEL
LIN {X 0,Y 247.899,Z 486.592,A -85,B 0,C 180,E1 -29484.841,E2 -29484.841} C_VEL
LIN {X 0,Y 250.616,Z 472.667,A -85,B 0,C 180,E1 -29485.741,E2 -29485.741} C_VEL
LIN {X 0,Y 252.424,Z 459.194,A -85,B 0,C 180,E1 -29486.344,E2 -29486.344} C_VEL
LIN {X 0,Y 255,Z 424.334,A -85,B 0,C 180,E1 -29487.262,E2 -29487.262} C_VEL
LIN {X 0,Y 255.679,Z 413.227,A -85,B 0,C 180,E1 -29487.564,E2 -29487.564} C_VEL
LIN {X 0,Y 249.581,Z 401.737,A -85,B 0,C 180,E1 -29489.89,E2 -29489.89} C_VEL
LIN {X 0,Y 244.116,Z 392.426,A -85,B 0,C 180,E1 -29492.15,E2 -29492.15} C_VEL
LIN {X 0,Y 237.746,Z 382.478,A -85,B 0,C 180,E1 -29495.06,E2 -29495.06} C_VEL
LIN {X 0,Y 232.016,Z 374.303,A -85,B 0,C 180,E1 -29498.032,E2 -29498.032} C_VEL
LIN {X 0,Y 228.81,Z 369.955,A -85,B 0,C 180,E1 -29499.885,E2 -29499.885} C_VEL
LIN {X 0,Y 225.623,Z 365.644,A -85,B 0,C 180,E1 -29501.914,E2 -29501.914} C_VEL
LIN {X 0,Y 222.905,Z 362.178,A -85,B 0,C 180,E1 -29503.814,E2 -29503.814} C_VEL
LIN {X 0,Y 222.023,Z 361.052,A -85,B 0,C 180,E1 -29504.475,E2 -29504.475} C_VEL
LIN {X 0,Y 219.417,Z 358.112,A -85,B 0,C 180,E1 -29506.548,E2 -29506.548} C_VEL
LIN {X 0,Y 218.126,Z 355.988,A -85,B 0,C 180,E1 -29507.746,E2 -29507.746} C_VEL
LIN {X 0,Y 215.537,Z 353.652,A -85,B 0,C 180,E1 -29510.262,E2 -29510.262} C_VEL
LIN {X 0,Y 213.817,Z 350.458,A -85,B 0,C 180,E1 -29512.471,E2 -29512.471} C_VEL
LIN {X 0,Y 211.107,Z 348.324,A -85,B 0,C 180,E1 -29516.493,E2 -29516.493} C_VEL
LIN {X 0,Y 209.798,Z 345.609,A -85,B 0,C 180,E1 -29519.851,E2 -29519.851} C_VEL
LIN {X 0,Y 209.609,Z 344.716,A -85,B 0,C 180,E1 -29520.709,E2 -29520.709} C_VEL
LIN {X 0,Y 209.068,Z 344.781,A -85,B 0,C 180,E1 -29528.429,E2 -29528.429} C_VEL
LIN {X 0,Y 209.512,Z 345.971,A -85,B 0,C 180,E1 -29530.718,E2 -29530.718} C_VEL
LIN {X 0,Y 211.666,Z 349.789,A -85,B 0,C 180,E1 -29535.923,E2 -29535.923} C_VEL
LIN {X 0,Y 215.194,Z 354.411,A -85,B 0,C 180,E1 -29540.756,E2 -29540.756} C_VEL
LIN {X 0,Y 219.758,Z 361.072,A -85,B 0,C 180,E1 -29545.234,E2 -29545.234} C_VEL
LIN {X 0,Y 224.805,Z 368.865,A -85,B 0,C 180,E1 -29549.121,E2 -29549.121} C_VEL
LIN {X 0,Y 228.659,Z 374.946,A -85,B 0,C 180,E1 -29551.64,E2 -29551.64} C_VEL
LIN {X 0,Y 232.456,Z 381.403,A -85,B 0,C 180,E1 -29553.88,E2 -29553.88} C_VEL
LIN {X 0,Y 237.201,Z 389.779,A -85,B 0,C 180,E1 -29556.396,E2 -29556.396} C_VEL
LIN {X 0,Y 242.443,Z 400.098,A -85,B 0,C 180,E1 -29558.917,E2 -29558.917} C_VEL
LIN {X 0,Y 247.932,Z 411.786,A -85,B 0,C 180,E1 -29561.329,E2 -29561.329} C_VEL
LIN {X 0,Y 253.087,Z 424.665,A -85,B 0,C 180,E1 -29563.467,E2 -29563.467} C_VEL
LIN {X 0,Y 253.854,Z 426.778,A -85,B 0,C 180,E1 -29563.777,E2 -29563.777} C_VEL
LIN {X 0,Y 254.361,Z 435.047,A -85,B 0,C 180,E1 -29564.284,E2 -29564.284} C_VEL
LIN {X 0,Y 251.251,Z 477.209,A -85,B 0,C 180,E1 -29565.349,E2 -29565.349} C_VEL
LIN {X 0,Y 249.127,Z 491.519,A -85,B 0,C 180,E1 -29565.91,E2 -29565.91} C_VEL
LIN {X 0,Y 246.337,Z 504.872,A -85,B 0,C 180,E1 -29566.694,E2 -29566.694} C_VEL
LIN {X 0,Y 242.842,Z 517.122,A -85,B 0,C 180,E1 -29567.613,E2 -29567.613} C_VEL
LIN {X 0,Y 238.881,Z 528.564,A -85,B 0,C 180,E1 -29568.726,E2 -29568.726} C_VEL
LIN {X 0,Y 236.231,Z 535.427,A -85,B 0,C 180,E1 -29569.561,E2 -29569.561} C_VEL
LIN {X 0,Y 233.721,Z 540.339,A -85,B 0,C 180,E1 -29570.124,E2 -29570.124} C_VEL
LIN {X 0,Y 228.03,Z 547.981,A -85,B 0,C 180,E1 -29570.835,E2 -29570.835} C_VEL
LIN {X 0,Y 222.169,Z 555.174,A -85,B 0,C 180,E1 -29571.672,E2 -29571.672} C_VEL
LIN {X 0,Y 219.363,Z 559.338,A -85,B 0,C 180,E1 -29572.452,E2 -29572.452} C_VEL
LIN {X 0,Y 213.518,Z 569.214,A -85,B 0,C 180,E1 -29574.971,E2 -29574.971} C_VEL
LIN {X 0,Y 207.516,Z 578.086,A -85,B 0,C 180,E1 -29577.891,E2 -29577.891} C_VEL
LIN {X 0,Y 202.202,Z 585.303,A -85,B 0,C 180,E1 -29580.996,E2 -29580.996} C_VEL
LIN {X 0,Y 197.018,Z 591.835,A -85,B 0,C 180,E1 -29584.752,E2 -29584.752} C_VEL
LIN {X 0,Y 192.992,Z 596.785,A -85,B 0,C 180,E1 -29588.725,E2 -29588.725} C_VEL
LIN {X 0,Y 189.868,Z 600.284,A -85,B 0,C 180,E1 -29592.84,E2 -29592.84} C_VEL
LIN {X 0,Y 187.769,Z 602.437,A -85,B 0,C 180,E1 -29597.072,E2 -29597.072} C_VEL
LIN {X 0,Y 186.669,Z 603.291,A -85,B 0,C 180,E1 -29601.373,E2 -29601.373} C_VEL
LIN {X 0,Y 186.672,Z 602.864,A -85,B 0,C 180,E1 -29605.701,E2 -29605.701} C_VEL
LIN {X 0,Y 187.572,Z 601.129,A -85,B 0,C 180,E1 -29610.005,E2 -29610.005} C_VEL
LIN {X 0,Y 188.181,Z 599.814,A -85,B 0,C 180,E1 -29612.138,E2 -29612.138} C_VEL
LIN {X 0,Y 187.714,Z 604.815,A -85,B 0,C 180,E1 -29615.358,E2 -29615.358} C_VEL
LIN {X 0,Y 187.767,Z 610.053,A -85,B 0,C 180,E1 -29619.669,E2 -29619.669} C_VEL
LIN {X 0,Y 188.65,Z 613.102,A -85,B 0,C 180,E1 -29622.877,E2 -29622.877} C_VEL
LIN {X 0,Y 190.975,Z 616.139,A -85,B 0,C 180,E1 -29627.068,E2 -29627.068} C_VEL
LIN {X 0,Y 194.414,Z 618,A -85,B 0,C 180,E1 -29631.123,E2 -29631.123} C_VEL
LIN {X 0,Y 198.99,Z 618.731,A -85,B 0,C 180,E1 -29634.991,E2 -29634.991} C_VEL
